(* IEC 61131-3 sources: SRCI/RobotLibrary/Library/POUs/AdvancedMove/MC_MoveCircularAbsolute, 1 file *)

(* ---- MC_MoveCircularAbsoluteFB.st ---- *)
/// Move the TCP to an absolute cartesian position (circular interpolation)
FUNCTION_BLOCK MC_MoveCircularAbsoluteFB EXTENDS RobotLibraryBaseExecuteFB
// -------------------------------------------------------------------------
//  SRCI Robot Library
// -------------------------------------------------------------------------
//
//  Object:      MoveCircularAbsoluteFB
//  Author:      Thorsten Brach
//  Date:        2024-06-01
//
//  Description:
//
//
//  Copyright:
//    (C) 2024 Thorsten Brach. All rights reserved
//             Licensed under the LGPL-3.0 license.
//
//  Disclaimer:
//    This project is provided without any guarantee and can be used for
//    private and commercial purposes. Any use is at the user’s
//    own risk and responsibility.
//
// -------------------------------------------------------------------------
VAR_INPUT
  /// Parameter which determines the behavior towards the previously sent and still active or buffered commands
  AbortingMode       : AbortingMode;
  /// Defines the target sequence in which the command will be executed
  SequenceFlag       : SequenceFlag;
  /// command results
  ParCmd             : MoveCircularAbsoluteParCmd;
END_VAR

VAR_OUTPUT
  /// Command is transferred and confirmed by the RC
  CommandBuffered    : BOOL;
  /// The command takes control of the motion of the according axis group
  Active             : BOOL;
  /// The command was aborted by another command.
  CommandAborted     : BOOL;
  /// TRUE, while command is interrupted during execution and can be continued
  CommandInterrupted : BOOL;
  /// command results
  OutCmd             : MoveCircularAbsoluteOutCmd;
END_VAR

VAR
  /// internal copy of command parameter
 _parCmd             : MoveCircularAbsoluteParCmd;
  /// command data to send
 _command            : MoveCircularAbsoluteSendData;
  /// response data received
 _response           : MoveCircularAbsoluteRecvData;
END_VAR

  SUPER^(AxesGroup := AxesGroup);

END_FUNCTION_BLOCK

METHOD INTERNAL CheckAddParameter : BOOL
VAR_INPUT
  /// Payload pointer
  PayloadPtr : UDINT;
END_VAR
VAR
  /// Payload as byte array
  Payload    : ARRAY [1..SIZEOF(_command)] OF BYTE;
  /// Null Byte array
  Null       : ARRAY [1..SIZEOF(_command)] OF BYTE;
  /// Data length to compare
  DataLen    : UDINT;
END_VAR

  // Payload pointer must be decreased by one byte, because ADR(Payload) is already one byte !
  PayloadPtr := LIMIT (0, PayloadPtr - 1, SIZEOF(Payload) -1);
  // Convert command struct to payload array
  SysDepMemCpy( pDest := ADR(Payload), pSrc := ADR(_command), DataLen := SIZEOF(_command));
  // Calculate the data length to compare - at least one byte must be compared !
  DataLen := LIMIT(1, SIZEOF(Payload) - PayloadPtr, SIZEOF(Payload));
  // Compare Payload-Array with Null-Byte-Array
  CheckAddParameter := SysDepMemCmp( pData1 := ADR(Payload) + PayloadPtr , pData2 := ADR(Null), DataLen := DataLen) <>  RobotLibraryConstants.OK ;

END_METHOD

METHOD PROTECTED CheckFunctionSupported : BOOL
VAR_IN_OUT
  /// Robot assignment of function
  AxesGroup : AxesGroup;
END_VAR

  CheckFunctionSupported := AxesGroup.State.RobotData.RCSupportedFunctions.MoveCircularAbsolute;

  IF ( NOT CheckFunctionSupported )
  THEN
    // call base implementation for set error and create log entry
    SUPER^.CheckFunctionSupported(AxesGroup := AxesGroup);
  END_IF

END_METHOD

METHOD PROTECTED CheckParameterChanged : BOOL
VAR_IN_OUT
  /// Robot assignment of function
  AxesGroup    : AxesGroup;
END_VAR

  // Check ParCmd Size is > 0, because MemCmp does not work correctly with size = 0
  IF (SIZEOF(ParCmd) = 0) OR (_stepCmd = 0)
  THEN
    RETURN;
  END_IF

  // compare memory
  _parameterChanged := ( SysDepMemCmp(pData1 := ADR(ParCmd), pData2 := ADR(_parCmd), DataLen := SIZEOF(ParCmd)) <> RobotLibraryConstants.OK );

  // check parameter valid ?
  _parameterValid   := CheckParameterValid( AxesGroup := AxesGroup );

  IF ((  _parameterChanged        )  AND
      (  _parameterValid          )) OR
      (  _parameterUpdateInternal )
  THEN
    // reset internal flag for send parameter update
   _parameterUpdateInternal := FALSE;
    // update internal copy of parameters
   _parCmd := ParCmd;
    // inc parameter sequence
   _command.ParSeq := _command.ParSeq + 1;
    // update command data
    CommandData := CreateCommandPayload(AxesGroup := AxesGroup); // ( Access via reference to rCommandFB in ACR )
    // notify active command register
    AxesGroup.Acyclic.ActiveCommandRegister.NotifyParameterChanged := _uniqueID;
  END_IF

END_METHOD

METHOD PROTECTED CheckParameterValid : BOOL
VAR_IN_OUT
  /// Robot assignment of function
  AxesGroup : AxesGroup;
END_VAR
VAR
  /// internal index for loops
 _idx : DINT;
END_VAR

  CheckParameterValid := TRUE;

  // Check AbortingMode valid ?
  IF (( AbortingMode <> AbortingModeEnum.BUFFER ) AND
      ( AbortingMode <> AbortingModeEnum.ABORT  ))
  THEN
    // Parameter not valid
    CheckParameterValid := FALSE;
    // Set error
    ErrorID := RobotLibraryErrorIdEnum.ERR_ABORTINGMODE_INVALID;
    // Create log entry
    CreateLogMessagePara1 ( Timestamp   := AxesGroup.State.SystemTime,
                            MessageType := MessageType.CMD,
                            Severity    := Severity.ERROR,
                            MessageCode := ErrorID,
                            MessageText := 'Invalid Parameter AbortingMode = {1}',
                            Para1       := ABORTING_MODE_TO_STRING(AbortingMode));
    RETURN;
  END_IF

  // Check SequenceFlag valid ?
  IF (( SequenceFlag <> SequenceFlagEnum.PRIMARY_SEQUENCE   ) AND
      ( SequenceFlag <> SequenceFlagEnum.SECONDARY_SEQUENCE ))
  THEN
    // Parameter not valid
    CheckParameterValid := FALSE;
    // Set error
    ErrorID := RobotLibraryErrorIdEnum.ERR_SEQFLAG_NOT_ALLOWED;
    // Create log entry
    CreateLogMessagePara1 ( Timestamp   := AxesGroup.State.SystemTime,
                            MessageType := MessageType.CMD,
                            Severity    := Severity.ERROR,
                            MessageCode := ErrorID,
                            MessageText := 'Invalid Parameter SequenceFlag = {1}',
                            Para1       := SEQUENCE_FLAG_TO_STRING(SequenceFlag));
    RETURN;
  END_IF

  // Check ParCmd.CircMode valid ?
  IF (( ParCmd.CircMode <> CircMode.BORDER            ) AND
      ( ParCmd.CircMode <> CircMode.CENTER            ) AND
      ( ParCmd.CircMode <> CircMode.CENTER_WITH_ANGLE ) AND
      ( ParCmd.CircMode <> CircMode.RADIUS            ))
  THEN
    // Parameter not valid
    CheckParameterValid := FALSE;
    // Set error
    ErrorID := RobotLibraryErrorIdEnum.ERR_INVALID_PAR_CMD;
    // Create log entry
    CreateLogMessagePara1 ( Timestamp   := AxesGroup.State.SystemTime,
                            MessageType := MessageType.CMD,
                            Severity    := Severity.ERROR,
                            MessageCode := ErrorID,
                            MessageText := 'Invalid Parameter ParCmd.CircMode = {1}',
                            Para1       :=  CIRC_MODE_TO_STRING(ParCmd.CircMode));
    RETURN;
  END_IF

  // Check ParCmd.AuxPoint.X valid ?
  IF ( SysDepIsValidReal(ParCmd.AuxPoint.X) = FALSE )
  THEN
    // Parameter not valid
    CheckParameterValid := FALSE;
    // Set error
    ErrorID := RobotLibraryErrorIdEnum.ERR_INVALID_PAR_CMD;

    // Create log entry
    CreateLogMessagePara1 ( Timestamp   := AxesGroup.State.SystemTime,
                            MessageType := MessageType.CMD,
                            Severity    := Severity.ERROR,
                            MessageCode := ErrorID,
                            MessageText := 'Invalid Parameter ParCmd.AuxPoint.X = {1}',
                            Para1       := VALID_REAL_TO_STRING(ParCmd.AuxPoint.X));
    RETURN;
  END_IF

  // Check ParCmd.AuxPoint.Y valid ?
  IF ( SysDepIsValidReal(ParCmd.AuxPoint.Y) = FALSE )
  THEN
    // Parameter not valid
    CheckParameterValid := FALSE;
    // Set error
    ErrorID := RobotLibraryErrorIdEnum.ERR_INVALID_PAR_CMD;

    // Create log entry
    CreateLogMessagePara1 ( Timestamp   := AxesGroup.State.SystemTime,
                            MessageType := MessageType.CMD,
                            Severity    := Severity.ERROR,
                            MessageCode := ErrorID,
                            MessageText := 'Invalid Parameter ParCmd.AuxPoint.Y = {1}',
                            Para1       := VALID_REAL_TO_STRING(ParCmd.AuxPoint.Y));
    RETURN;
  END_IF

  // Check ParCmd.AuxPoint.Z valid ?
  IF ( SysDepIsValidReal(ParCmd.AuxPoint.Z) = FALSE )
  THEN
    // Parameter not valid
    CheckParameterValid := FALSE;
    // Set error
    ErrorID := RobotLibraryErrorIdEnum.ERR_INVALID_PAR_CMD;

    // Create log entry
    CreateLogMessagePara1 ( Timestamp   := AxesGroup.State.SystemTime,
                            MessageType := MessageType.CMD,
                            Severity    := Severity.ERROR,
                            MessageCode := ErrorID,
                            MessageText := 'Invalid Parameter ParCmd.AuxPoint.Z = {1}',
                            Para1       := VALID_REAL_TO_STRING(ParCmd.AuxPoint.Z));
    RETURN;
  END_IF

  // Check ParCmd.AuxPoint.Rx valid ?
  IF ( SysDepIsValidReal(ParCmd.AuxPoint.Rx) = FALSE )
  THEN
    // Parameter not valid
    CheckParameterValid := FALSE;
    // Set error
    ErrorID := RobotLibraryErrorIdEnum.ERR_INVALID_PAR_CMD;

    // Create log entry
    CreateLogMessagePara1 ( Timestamp   := AxesGroup.State.SystemTime,
                            MessageType := MessageType.CMD,
                            Severity    := Severity.ERROR,
                            MessageCode := ErrorID,
                            MessageText := 'Invalid Parameter ParCmd.AuxPoint.Rx = {1}',
                            Para1       := VALID_REAL_TO_STRING(ParCmd.AuxPoint.Rx));
    RETURN;
  END_IF

  // Check ParCmd.AuxPoint.Ry valid ?
  IF ( SysDepIsValidReal(ParCmd.AuxPoint.Ry) = FALSE )
  THEN
    // Parameter not valid
    CheckParameterValid := FALSE;
    // Set error
    ErrorID := RobotLibraryErrorIdEnum.ERR_INVALID_PAR_CMD;

    // Create log entry
    CreateLogMessagePara1 ( Timestamp   := AxesGroup.State.SystemTime,
                            MessageType := MessageType.CMD,
                            Severity    := Severity.ERROR,
                            MessageCode := ErrorID,
                            MessageText := 'Invalid Parameter ParCmd.AuxPoint.Ry = {1}',
                            Para1       := VALID_REAL_TO_STRING(ParCmd.AuxPoint.Ry));
    RETURN;
  END_IF

  // Check ParCmd.AuxPoint.Rz valid ?
  IF ( SysDepIsValidReal(ParCmd.AuxPoint.Rz) = FALSE )
  THEN
    // Parameter not valid
    CheckParameterValid := FALSE;
    // Set error
    ErrorID := RobotLibraryErrorIdEnum.ERR_INVALID_PAR_CMD;

    // Create log entry
    CreateLogMessagePara1 ( Timestamp   := AxesGroup.State.SystemTime,
                            MessageType := MessageType.CMD,
                            Severity    := Severity.ERROR,
                            MessageCode := ErrorID,
                            MessageText := 'Invalid Parameter ParCmd.AuxPoint.Rz = {1}',
                            Para1       := VALID_REAL_TO_STRING(ParCmd.AuxPoint.Rz));
    RETURN;
  END_IF

  // Check ParCmd.AuxPoint.E1 valid ?
  IF ( SysDepIsValidReal(ParCmd.AuxPoint.E1) = FALSE )
  THEN
    // Parameter not valid
    CheckParameterValid := FALSE;
    // Set error
    ErrorID := RobotLibraryErrorIdEnum.ERR_INVALID_PAR_CMD;

    // Create log entry
    CreateLogMessagePara1 ( Timestamp   := AxesGroup.State.SystemTime,
                            MessageType := MessageType.CMD,
                            Severity    := Severity.ERROR,
                            MessageCode := ErrorID,
                            MessageText := 'Invalid Parameter ParCmd.AuxPoint.E1 = {1}',
                            Para1       := VALID_REAL_TO_STRING(ParCmd.AuxPoint.E1));
    RETURN;
  END_IF

  // Check ParCmd.AuxPoint.E2 valid ?
  IF ( SysDepIsValidReal(ParCmd.AuxPoint.E2) = FALSE )
  THEN
    // Parameter not valid
    CheckParameterValid := FALSE;
    // Set error
    ErrorID := RobotLibraryErrorIdEnum.ERR_INVALID_PAR_CMD;

    // Create log entry
    CreateLogMessagePara1 ( Timestamp   := AxesGroup.State.SystemTime,
                            MessageType := MessageType.CMD,
                            Severity    := Severity.ERROR,
                            MessageCode := ErrorID,
                            MessageText := 'Invalid Parameter ParCmd.AuxPoint.E2 = {1}',
                            Para1       := VALID_REAL_TO_STRING(ParCmd.AuxPoint.E2));
    RETURN;
  END_IF

  // Check ParCmd.AuxPoint.E3 valid ?
  IF ( SysDepIsValidReal(ParCmd.AuxPoint.E3) = FALSE )
  THEN
    // Parameter not valid
    CheckParameterValid := FALSE;
    // Set error
    ErrorID := RobotLibraryErrorIdEnum.ERR_INVALID_PAR_CMD;

    // Create log entry
    CreateLogMessagePara1 ( Timestamp   := AxesGroup.State.SystemTime,
                            MessageType := MessageType.CMD,
                            Severity    := Severity.ERROR,
                            MessageCode := ErrorID,
                            MessageText := 'Invalid Parameter ParCmd.AuxPoint.E3 = {1}',
                            Para1       := VALID_REAL_TO_STRING(ParCmd.AuxPoint.E3));
    RETURN;
  END_IF

  // Check ParCmd.AuxPoint.E4 valid ?
  IF ( SysDepIsValidReal(ParCmd.AuxPoint.E4) = FALSE )
  THEN
    // Parameter not valid
    CheckParameterValid := FALSE;
    // Set error
    ErrorID := RobotLibraryErrorIdEnum.ERR_INVALID_PAR_CMD;

    // Create log entry
    CreateLogMessagePara1 ( Timestamp   := AxesGroup.State.SystemTime,
                            MessageType := MessageType.CMD,
                            Severity    := Severity.ERROR,
                            MessageCode := ErrorID,
                            MessageText := 'Invalid Parameter ParCmd.AuxPoint.E4 = {1}',
                            Para1       := VALID_REAL_TO_STRING(ParCmd.AuxPoint.E4));
    RETURN;
  END_IF

  // Check ParCmd.AuxPoint.E5 valid ?
  IF ( SysDepIsValidReal(ParCmd.AuxPoint.E5) = FALSE )
  THEN
    // Parameter not valid
    CheckParameterValid := FALSE;
    // Set error
    ErrorID := RobotLibraryErrorIdEnum.ERR_INVALID_PAR_CMD;

    // Create log entry
    CreateLogMessagePara1 ( Timestamp   := AxesGroup.State.SystemTime,
                            MessageType := MessageType.CMD,
                            Severity    := Severity.ERROR,
                            MessageCode := ErrorID,
                            MessageText := 'Invalid Parameter ParCmd.AuxPoint.E5 = {1}',
                            Para1       := VALID_REAL_TO_STRING(ParCmd.AuxPoint.E5));
    RETURN;
  END_IF

  // Check ParCmd.AuxPoint.E6 valid ?
  IF ( SysDepIsValidReal(ParCmd.AuxPoint.E6) = FALSE )
  THEN
    // Parameter not valid
    CheckParameterValid := FALSE;
    // Set error
    ErrorID := RobotLibraryErrorIdEnum.ERR_INVALID_PAR_CMD;

    // Create log entry
    CreateLogMessagePara1 ( Timestamp   := AxesGroup.State.SystemTime,
                            MessageType := MessageType.CMD,
                            Severity    := Severity.ERROR,
                            MessageCode := ErrorID,
                            MessageText := 'Invalid Parameter ParCmd.AuxPoint.E6 = {1}',
                            Para1       := VALID_REAL_TO_STRING(ParCmd.AuxPoint.E6));
    RETURN;
  END_IF

  // Check ParCmd.AuxPoint.Config.Shoulder valid ?
  IF (( ParCmd.AuxPoint.Config.Shoulder <> ArmConfigShoulder.USE_CONFIG ) AND
      ( ParCmd.AuxPoint.Config.Shoulder <> ArmConfigShoulder.SAME       ) AND
      ( ParCmd.AuxPoint.Config.Shoulder <> ArmConfigShoulder.FREE       ) AND
      ( ParCmd.AuxPoint.Config.Shoulder <> ArmConfigShoulder.BACK       ) AND
      ( ParCmd.AuxPoint.Config.Shoulder <> ArmConfigShoulder.FRONT      ))
  THEN
    // Parameter not valid
    CheckParameterValid := FALSE;
    // Set error
    ErrorID := RobotLibraryErrorIdEnum.ERR_CONFIGMODE_SHOULDER_INVALID;
    // Create log entry
    CreateLogMessagePara1 ( Timestamp   := AxesGroup.State.SystemTime,
                            MessageType := MessageType.CMD,
                            Severity    := Severity.ERROR,
                            MessageCode := ErrorID,
                            MessageText := 'Invalid Parameter ParCmd.AuxPoint.Config.Shoulder = {1}',
                            Para1       :=  ARM_CONFIG_SHOULDER_TO_STRING(ParCmd.AuxPoint.Config.Shoulder));
    RETURN;
  END_IF

  // Check ParCmd.AuxPoint.Config.Elbow valid ?
  IF (( ParCmd.AuxPoint.Config.Elbow <> ArmConfigElbow.USE_CONFIG ) AND
      ( ParCmd.AuxPoint.Config.Elbow <> ArmConfigElbow.SAME       ) AND
      ( ParCmd.AuxPoint.Config.Elbow <> ArmConfigElbow.FREE       ) AND
      ( ParCmd.AuxPoint.Config.Elbow <> ArmConfigElbow.DOWN       ) AND
      ( ParCmd.AuxPoint.Config.Elbow <> ArmConfigElbow.UP         ))
  THEN
    // Parameter not valid
    CheckParameterValid := FALSE;
    // Set error
    ErrorID := RobotLibraryErrorIdEnum.ERR_CONFIGMODE_ELBOW_INVALID;
    // Create log entry
    CreateLogMessagePara1 ( Timestamp   := AxesGroup.State.SystemTime,
                            MessageType := MessageType.CMD,
                            Severity    := Severity.ERROR,
                            MessageCode := ErrorID,
                            MessageText := 'Invalid Parameter ParCmd.AuxPoint.Config.Elbow = {1}',
                            Para1       :=  ARM_CONFIG_ELBOW_TO_STRING(ParCmd.AuxPoint.Config.Elbow));
    RETURN;
  END_IF

  // Check ParCmd.AuxPoint.Config.Wrist valid ?
  IF (( ParCmd.AuxPoint.Config.Wrist <> ArmConfigWrist.USE_CONFIG ) AND
      ( ParCmd.AuxPoint.Config.Wrist <> ArmConfigWrist.SAME       ) AND
      ( ParCmd.AuxPoint.Config.Wrist <> ArmConfigWrist.FREE       ) AND
      ( ParCmd.AuxPoint.Config.Wrist <> ArmConfigWrist.FLIP       ) AND
      ( ParCmd.AuxPoint.Config.Wrist <> ArmConfigWrist.NON_FLIP   ))
  THEN
    // Parameter not valid
    CheckParameterValid := FALSE;
    // Set error
    ErrorID := RobotLibraryErrorIdEnum.ERR_CONFIGMODE_WRIST_INVALID;
    // Create log entry
    CreateLogMessagePara1 ( Timestamp   := AxesGroup.State.SystemTime,
                            MessageType := MessageType.CMD,
                            Severity    := Severity.ERROR,
                            MessageCode := ErrorID,
                            MessageText := 'Invalid Parameter ParCmd.AuxPoint.Config.Wrist = {1}',
                            Para1       :=  ARM_CONFIG_WRIST_TO_STRING(ParCmd.AuxPoint.Config.Wrist));
    RETURN;
  END_IF

  // Check ParCmd.CircPlane valid ?
  IF (( ParCmd.CircPlane <> CircPlane.XZ_PLANE ) AND
      ( ParCmd.CircPlane <> CircPlane.YZ_PLANE ) AND
      ( ParCmd.CircPlane <> CircPlane.XY_PLANE ))
  THEN
    // Parameter not valid
    CheckParameterValid := FALSE;
    // Set error
    ErrorID := RobotLibraryErrorIdEnum.ERR_INVALID_PAR_CMD;
    // Create log entry
    CreateLogMessagePara1 ( Timestamp   := AxesGroup.State.SystemTime,
                            MessageType := MessageType.CMD,
                            Severity    := Severity.ERROR,
                            MessageCode := ErrorID,
                            MessageText := 'Invalid Parameter ParCmd.CircPlane = {1}',
                            Para1       :=  CIRC_PLANE_TO_STRING(ParCmd.CircPlane));
    RETURN;
  END_IF

  // Check ParCmd.Tolerance valid ?
  IF ( SysDepIsValidReal(ParCmd.Tolerance) = FALSE )
  THEN
    // Parameter not valid
    CheckParameterValid := FALSE;
    // Set error
    ErrorID := RobotLibraryErrorIdEnum.ERR_INVALID_PAR_CMD;

    // Create log entry
    CreateLogMessagePara1 ( Timestamp   := AxesGroup.State.SystemTime,
                            MessageType := MessageType.CMD,
                            Severity    := Severity.ERROR,
                            MessageCode := ErrorID,
                            MessageText := 'Invalid Parameter ParCmd.Tolerance = {1}',
                            Para1       := VALID_REAL_TO_STRING(ParCmd.Tolerance));
    RETURN;
  END_IF

  // Check ParCmd.EndPoint.X valid ?
  IF ( SysDepIsValidReal(ParCmd.EndPoint.X) = FALSE )
  THEN
    // Parameter not valid
    CheckParameterValid := FALSE;
    // Set error
    ErrorID := RobotLibraryErrorIdEnum.ERR_INVALID_PAR_CMD;

    // Create log entry
    CreateLogMessagePara1 ( Timestamp   := AxesGroup.State.SystemTime,
                            MessageType := MessageType.CMD,
                            Severity    := Severity.ERROR,
                            MessageCode := ErrorID,
                            MessageText := 'Invalid Parameter ParCmd.EndPoint.X = {1}',
                            Para1       := VALID_REAL_TO_STRING(ParCmd.EndPoint.X));
    RETURN;
  END_IF

  // Check ParCmd.EndPoint.Y valid ?
  IF ( SysDepIsValidReal(ParCmd.EndPoint.Y) = FALSE )
  THEN
    // Parameter not valid
    CheckParameterValid := FALSE;
    // Set error
    ErrorID := RobotLibraryErrorIdEnum.ERR_INVALID_PAR_CMD;

    // Create log entry
    CreateLogMessagePara1 ( Timestamp   := AxesGroup.State.SystemTime,
                            MessageType := MessageType.CMD,
                            Severity    := Severity.ERROR,
                            MessageCode := ErrorID,
                            MessageText := 'Invalid Parameter ParCmd.EndPoint.Y = {1}',
                            Para1       := VALID_REAL_TO_STRING(ParCmd.EndPoint.Y));
    RETURN;
  END_IF

  // Check ParCmd.EndPoint.Z valid ?
  IF ( SysDepIsValidReal(ParCmd.EndPoint.Z) = FALSE )
  THEN
    // Parameter not valid
    CheckParameterValid := FALSE;
    // Set error
    ErrorID := RobotLibraryErrorIdEnum.ERR_INVALID_PAR_CMD;

    // Create log entry
    CreateLogMessagePara1 ( Timestamp   := AxesGroup.State.SystemTime,
                            MessageType := MessageType.CMD,
                            Severity    := Severity.ERROR,
                            MessageCode := ErrorID,
                            MessageText := 'Invalid Parameter ParCmd.EndPoint.Z = {1}',
                            Para1       := VALID_REAL_TO_STRING(ParCmd.EndPoint.Z));
    RETURN;
  END_IF

  // Check ParCmd.EndPoint.Rx valid ?
  IF ( SysDepIsValidReal(ParCmd.EndPoint.Rx) = FALSE )
  THEN
    // Parameter not valid
    CheckParameterValid := FALSE;
    // Set error
    ErrorID := RobotLibraryErrorIdEnum.ERR_INVALID_PAR_CMD;

    // Create log entry
    CreateLogMessagePara1 ( Timestamp   := AxesGroup.State.SystemTime,
                            MessageType := MessageType.CMD,
                            Severity    := Severity.ERROR,
                            MessageCode := ErrorID,
                            MessageText := 'Invalid Parameter ParCmd.EndPoint.Rx = {1}',
                            Para1       := VALID_REAL_TO_STRING(ParCmd.EndPoint.Rx));
    RETURN;
  END_IF

  // Check ParCmd.EndPoint.Ry valid ?
  IF ( SysDepIsValidReal(ParCmd.EndPoint.Ry) = FALSE )
  THEN
    // Parameter not valid
    CheckParameterValid := FALSE;
    // Set error
    ErrorID := RobotLibraryErrorIdEnum.ERR_INVALID_PAR_CMD;

    // Create log entry
    CreateLogMessagePara1 ( Timestamp   := AxesGroup.State.SystemTime,
                            MessageType := MessageType.CMD,
                            Severity    := Severity.ERROR,
                            MessageCode := ErrorID,
                            MessageText := 'Invalid Parameter ParCmd.EndPoint.Ry = {1}',
                            Para1       := VALID_REAL_TO_STRING(ParCmd.EndPoint.Ry));
    RETURN;
  END_IF

  // Check ParCmd.EndPoint.Rz valid ?
  IF ( SysDepIsValidReal(ParCmd.EndPoint.Rz) = FALSE )
  THEN
    // Parameter not valid
    CheckParameterValid := FALSE;
    // Set error
    ErrorID := RobotLibraryErrorIdEnum.ERR_INVALID_PAR_CMD;

    // Create log entry
    CreateLogMessagePara1 ( Timestamp   := AxesGroup.State.SystemTime,
                            MessageType := MessageType.CMD,
                            Severity    := Severity.ERROR,
                            MessageCode := ErrorID,
                            MessageText := 'Invalid Parameter ParCmd.EndPoint.Rz = {1}',
                            Para1       := VALID_REAL_TO_STRING(ParCmd.EndPoint.Rz));
    RETURN;
  END_IF

  // Check ParCmd.EndPoint.E1 valid ?
  IF ( SysDepIsValidReal(ParCmd.EndPoint.E1) = FALSE )
  THEN
    // Parameter not valid
    CheckParameterValid := FALSE;
    // Set error
    ErrorID := RobotLibraryErrorIdEnum.ERR_INVALID_PAR_CMD;

    // Create log entry
    CreateLogMessagePara1 ( Timestamp   := AxesGroup.State.SystemTime,
                            MessageType := MessageType.CMD,
                            Severity    := Severity.ERROR,
                            MessageCode := ErrorID,
                            MessageText := 'Invalid Parameter ParCmd.EndPoint.E1 = {1}',
                            Para1       := VALID_REAL_TO_STRING(ParCmd.EndPoint.E1));
    RETURN;
  END_IF

  // Check ParCmd.EndPoint.E2 valid ?
  IF ( SysDepIsValidReal(ParCmd.EndPoint.E2) = FALSE )
  THEN
    // Parameter not valid
    CheckParameterValid := FALSE;
    // Set error
    ErrorID := RobotLibraryErrorIdEnum.ERR_INVALID_PAR_CMD;

    // Create log entry
    CreateLogMessagePara1 ( Timestamp   := AxesGroup.State.SystemTime,
                            MessageType := MessageType.CMD,
                            Severity    := Severity.ERROR,
                            MessageCode := ErrorID,
                            MessageText := 'Invalid Parameter ParCmd.EndPoint.E2 = {1}',
                            Para1       := VALID_REAL_TO_STRING(ParCmd.EndPoint.E2));
    RETURN;
  END_IF

  // Check ParCmd.EndPoint.E3 valid ?
  IF ( SysDepIsValidReal(ParCmd.EndPoint.E3) = FALSE )
  THEN
    // Parameter not valid
    CheckParameterValid := FALSE;
    // Set error
    ErrorID := RobotLibraryErrorIdEnum.ERR_INVALID_PAR_CMD;

    // Create log entry
    CreateLogMessagePara1 ( Timestamp   := AxesGroup.State.SystemTime,
                            MessageType := MessageType.CMD,
                            Severity    := Severity.ERROR,
                            MessageCode := ErrorID,
                            MessageText := 'Invalid Parameter ParCmd.EndPoint.E3 = {1}',
                            Para1       := VALID_REAL_TO_STRING(ParCmd.EndPoint.E3));
    RETURN;
  END_IF

  // Check ParCmd.EndPoint.E4 valid ?
  IF ( SysDepIsValidReal(ParCmd.EndPoint.E4) = FALSE )
  THEN
    // Parameter not valid
    CheckParameterValid := FALSE;
    // Set error
    ErrorID := RobotLibraryErrorIdEnum.ERR_INVALID_PAR_CMD;

    // Create log entry
    CreateLogMessagePara1 ( Timestamp   := AxesGroup.State.SystemTime,
                            MessageType := MessageType.CMD,
                            Severity    := Severity.ERROR,
                            MessageCode := ErrorID,
                            MessageText := 'Invalid Parameter ParCmd.EndPoint.E4 = {1}',
                            Para1       := VALID_REAL_TO_STRING(ParCmd.EndPoint.E4));
    RETURN;
  END_IF

  // Check ParCmd.EndPoint.E5 valid ?
  IF ( SysDepIsValidReal(ParCmd.EndPoint.E5) = FALSE )
  THEN
    // Parameter not valid
    CheckParameterValid := FALSE;
    // Set error
    ErrorID := RobotLibraryErrorIdEnum.ERR_INVALID_PAR_CMD;

    // Create log entry
    CreateLogMessagePara1 ( Timestamp   := AxesGroup.State.SystemTime,
                            MessageType := MessageType.CMD,
                            Severity    := Severity.ERROR,
                            MessageCode := ErrorID,
                            MessageText := 'Invalid Parameter ParCmd.EndPoint.E5 = {1}',
                            Para1       := VALID_REAL_TO_STRING(ParCmd.EndPoint.E5));
    RETURN;
  END_IF

  // Check ParCmd.EndPoint.E6 valid ?
  IF ( SysDepIsValidReal(ParCmd.EndPoint.E6) = FALSE )
  THEN
    // Parameter not valid
    CheckParameterValid := FALSE;
    // Set error
    ErrorID := RobotLibraryErrorIdEnum.ERR_INVALID_PAR_CMD;

    // Create log entry
    CreateLogMessagePara1 ( Timestamp   := AxesGroup.State.SystemTime,
                            MessageType := MessageType.CMD,
                            Severity    := Severity.ERROR,
                            MessageCode := ErrorID,
                            MessageText := 'Invalid Parameter ParCmd.EndPoint.E6 = {1}',
                            Para1       := VALID_REAL_TO_STRING(ParCmd.EndPoint.E6));
    RETURN;
  END_IF

  // Check ParCmd.EndPoint.Config.Shoulder valid ?
  IF (( ParCmd.EndPoint.Config.Shoulder <> ArmConfigShoulder.USE_CONFIG ) AND
      ( ParCmd.EndPoint.Config.Shoulder <> ArmConfigShoulder.SAME       ) AND
      ( ParCmd.EndPoint.Config.Shoulder <> ArmConfigShoulder.FREE       ) AND
      ( ParCmd.EndPoint.Config.Shoulder <> ArmConfigShoulder.BACK       ) AND
      ( ParCmd.EndPoint.Config.Shoulder <> ArmConfigShoulder.FRONT      ))
  THEN
    // Parameter not valid
    CheckParameterValid := FALSE;
    // Set error
    ErrorID := RobotLibraryErrorIdEnum.ERR_CONFIGMODE_SHOULDER_INVALID;
    // Create log entry
    CreateLogMessagePara1 ( Timestamp   := AxesGroup.State.SystemTime,
                            MessageType := MessageType.CMD,
                            Severity    := Severity.ERROR,
                            MessageCode := ErrorID,
                            MessageText := 'Invalid Parameter ParCmd.EndPoint.Config.Shoulder = {1}',
                            Para1       :=  ARM_CONFIG_SHOULDER_TO_STRING(ParCmd.EndPoint.Config.Shoulder));
    RETURN;
  END_IF

  // Check ParCmd.EndPoint.Config.Elbow valid ?
  IF (( ParCmd.EndPoint.Config.Elbow <> ArmConfigElbow.USE_CONFIG ) AND
      ( ParCmd.EndPoint.Config.Elbow <> ArmConfigElbow.SAME       ) AND
      ( ParCmd.EndPoint.Config.Elbow <> ArmConfigElbow.FREE       ) AND
      ( ParCmd.EndPoint.Config.Elbow <> ArmConfigElbow.DOWN       ) AND
      ( ParCmd.EndPoint.Config.Elbow <> ArmConfigElbow.UP         ))
  THEN
    // Parameter not valid
    CheckParameterValid := FALSE;
    // Set error
    ErrorID := RobotLibraryErrorIdEnum.ERR_CONFIGMODE_ELBOW_INVALID;
    // Create log entry
    CreateLogMessagePara1 ( Timestamp   := AxesGroup.State.SystemTime,
                            MessageType := MessageType.CMD,
                            Severity    := Severity.ERROR,
                            MessageCode := ErrorID,
                            MessageText := 'Invalid Parameter ParCmd.EndPoint.Config.Elbow = {1}',
                            Para1       :=  ARM_CONFIG_ELBOW_TO_STRING(ParCmd.EndPoint.Config.Elbow));
    RETURN;
  END_IF

  // Check ParCmd.EndPoint.Config.Wrist valid ?
  IF (( ParCmd.EndPoint.Config.Wrist <> ArmConfigWrist.USE_CONFIG ) AND
      ( ParCmd.EndPoint.Config.Wrist <> ArmConfigWrist.SAME       ) AND
      ( ParCmd.EndPoint.Config.Wrist <> ArmConfigWrist.FREE       ) AND
      ( ParCmd.EndPoint.Config.Wrist <> ArmConfigWrist.FLIP       ) AND
      ( ParCmd.EndPoint.Config.Wrist <> ArmConfigWrist.NON_FLIP   ))
  THEN
    // Parameter not valid
    CheckParameterValid := FALSE;
    // Set error
    ErrorID := RobotLibraryErrorIdEnum.ERR_CONFIGMODE_WRIST_INVALID;
    // Create log entry
    CreateLogMessagePara1 ( Timestamp   := AxesGroup.State.SystemTime,
                            MessageType := MessageType.CMD,
                            Severity    := Severity.ERROR,
                            MessageCode := ErrorID,
                            MessageText := 'Invalid Parameter ParCmd.EndPoint.Config.Wrist = {1}',
                            Para1       :=  ARM_CONFIG_WRIST_TO_STRING(ParCmd.EndPoint.Config.Wrist));
    RETURN;
  END_IF

  // Check ParCmd.Angle valid ?
  IF ( SysDepIsValidReal(ParCmd.Angle) = FALSE )
  THEN
    // Parameter not valid
    CheckParameterValid := FALSE;
    // Set error
    ErrorID := RobotLibraryErrorIdEnum.ERR_INVALID_PAR_CMD;

    // Create log entry
    CreateLogMessagePara1 ( Timestamp   := AxesGroup.State.SystemTime,
                            MessageType := MessageType.CMD,
                            Severity    := Severity.ERROR,
                            MessageCode := ErrorID,
                            MessageText := 'Invalid Parameter ParCmd.Angle = {1}',
                            Para1       := VALID_REAL_TO_STRING(ParCmd.Angle));
    RETURN;
  END_IF

  // Check ParCmd.PathChoice valid ?
  IF (( ParCmd.PathChoice <> PathChoice.CLOCKWISE  ) AND
      ( ParCmd.PathChoice <> PathChoice.COUNTERCLOCKWISE ))
  THEN
    // Parameter not valid
    CheckParameterValid := FALSE;
    // Set error
    ErrorID := RobotLibraryErrorIdEnum.ERR_INVALID_PAR_CMD;
    // Create log entry
    CreateLogMessagePara1 ( Timestamp   := AxesGroup.State.SystemTime,
                            MessageType := MessageType.CMD,
                            Severity    := Severity.ERROR,
                            MessageCode := ErrorID,
                            MessageText := 'Invalid Parameter ParCmd.PathChoice = {1}',
                            Para1       := PATH_CHOICE_TO_STRING(ParCmd.PathChoice));
    RETURN;
  END_IF

  // Check ParCmd.VelocityRate valid ?
  IF  (( SysDepIsValidReal(ParCmd.VelocityRate) = FALSE )  OR
      ((                   ParCmd.VelocityRate  <     0 )  AND
       (                   ParCmd.VelocityRate <>    -1 )) OR
       (                   ParCmd.VelocityRate  >   100 ))
  THEN
    // Parameter not valid
    CheckParameterValid := FALSE;
    // Set error
    ErrorID := RobotLibraryErrorIdEnum.ERR_VELOCITY_INVALID;
    // Create log entry
    CreateLogMessagePara1 ( Timestamp   := AxesGroup.State.SystemTime,
                            MessageType := MessageType.CMD,
                            Severity    := Severity.ERROR,
                            MessageCode := ErrorID,
                            MessageText := 'Invalid Parameter ParCmd.VelocityRate = {1}',
                            Para1       := VALID_REAL_TO_STRING(ParCmd.VelocityRate));
    RETURN;
  END_IF

  // Check ParCmd.AccelerationRate valid ?
  IF  (( SysDepIsValidReal(ParCmd.AccelerationRate) = FALSE )  OR
      ((                   ParCmd.AccelerationRate  <     0 )  AND
       (                   ParCmd.AccelerationRate <>    -1 )) OR
       (                   ParCmd.AccelerationRate  >   100 ))
  THEN
    // Parameter not valid
    CheckParameterValid := FALSE;
    // Set error
    ErrorID := RobotLibraryErrorIdEnum.ERR_ACCELERATION_INVALID;
    // Create log entry
    CreateLogMessagePara1 ( Timestamp   := AxesGroup.State.SystemTime,
                            MessageType := MessageType.CMD,
                            Severity    := Severity.ERROR,
                            MessageCode := ErrorID,
                            MessageText := 'Invalid Parameter ParCmd.AccelerationRate = {1}',
                            Para1       := VALID_REAL_TO_STRING(ParCmd.AccelerationRate));
    RETURN;
  END_IF

  // Check ParCmd.DecelerationRate valid ?
  IF  (( SysDepIsValidReal(ParCmd.DecelerationRate) = FALSE )  OR
      ((                   ParCmd.DecelerationRate  <     0 )  AND
       (                   ParCmd.DecelerationRate <>    -1 )) OR
       (                   ParCmd.DecelerationRate  >   100 ))
  THEN
    // Parameter not valid
    CheckParameterValid := FALSE;
    // Set error
    ErrorID := RobotLibraryErrorIdEnum.ERR_DECELERATION_INVALID;
    // Create log entry
    CreateLogMessagePara1 ( Timestamp   := AxesGroup.State.SystemTime,
                            MessageType := MessageType.CMD,
                            Severity    := Severity.ERROR,
                            MessageCode := ErrorID,
                            MessageText := 'Invalid Parameter ParCmd.DecelerationRate = {1}',
                            Para1       := VALID_REAL_TO_STRING(ParCmd.DecelerationRate));
    RETURN;
  END_IF

  // Check ParCmd.JerkRate valid ?
  IF  (( SysDepIsValidReal(ParCmd.JerkRate) = FALSE )  OR
      ((                   ParCmd.JerkRate  <     0 )  AND
       (                   ParCmd.JerkRate <>    -1 )) OR
       (                   ParCmd.JerkRate  >   100 ))
  THEN
    // Parameter not valid
    CheckParameterValid := FALSE;
    // Set error
    ErrorID := RobotLibraryErrorIdEnum.ERR_JERK_INVALID;
    // Create log entry
    CreateLogMessagePara1 ( Timestamp   := AxesGroup.State.SystemTime,
                            MessageType := MessageType.CMD,
                            Severity    := Severity.ERROR,
                            MessageCode := ErrorID,
                            MessageText := 'Invalid Parameter ParCmd.JerkRate = {1}',
                            Para1       := VALID_REAL_TO_STRING(ParCmd.JerkRate));
    RETURN;
  END_IF

  // Check ParCmd.ToolNo valid ?
  IF (( ParCmd.ToolNo <   0                                                ) OR
      ( ParCmd.ToolNo > 254                                                ) OR
      ( ParCmd.ToolNo > AxesGroup.State.ConfigurationData.HighestToolIndex ) OR
      ( ParCmd.ToolNo > RobotLibraryParameter.TOOL_MAX -1                  ))
  THEN
    // Parameter not valid
    CheckParameterValid := FALSE;

    // Check ToolNo available on RC ?
    IF ( ParCmd.ToolNo > AxesGroup.State.ConfigurationData.HighestToolIndex )
    THEN
      ErrorID := RobotLibraryErrorIdEnum.ERR_TOOLNO_UNAVAILABLE;
    ELSE
      ErrorID := RobotLibraryErrorIdEnum.ERR_TOOLNO_RANGE;
  	END_IF

    // Create log entry
    CreateLogMessagePara1 ( Timestamp   := AxesGroup.State.SystemTime,
                            MessageType := MessageType.CMD,
                            Severity    := Severity.ERROR,
                            MessageCode := ErrorID,
                            MessageText := 'Invalid Parameter ParCmd.ToolNo = {1}',
                            Para1       := USINT_TO_STRING(ParCmd.ToolNo));
    RETURN;
  END_IF

  // Check ParCmd.FrameNo valid ?
  IF (( ParCmd.FrameNo <   0                                                 ) OR
      ( ParCmd.FrameNo > 254                                                 ) OR
      ( ParCmd.FrameNo > AxesGroup.State.ConfigurationData.HighestFrameIndex ) OR
      ( ParCmd.FrameNo > RobotLibraryParameter.FRAME_MAX -1                  ))
  THEN
    // Parameter not valid
    CheckParameterValid := FALSE;

    // Check FrameNo available on RC ?
    IF ( ParCmd.FrameNo > AxesGroup.State.ConfigurationData.HighestFrameIndex )
    THEN
      ErrorID := RobotLibraryErrorIdEnum.ERR_FRAMENO_UNAVAILABLE;
    ELSE
      ErrorID := RobotLibraryErrorIdEnum.ERR_FRAMENO_RANGE;
  	END_IF

    // Create log entry
    CreateLogMessagePara1 ( Timestamp   := AxesGroup.State.SystemTime,
                            MessageType := MessageType.CMD,
                            Severity    := Severity.ERROR,
                            MessageCode := ErrorID,
                            MessageText := 'Invalid Parameter ParCmd.FrameNo = {1}',
                            Para1       := USINT_TO_STRING(ParCmd.FrameNo));
    RETURN;
  END_IF

  // Check ParCmd.BlendingMode valid ?
  IF (( ParCmd.BlendingMode <> BlendingMode.EXACT_STOP           ) AND
      ( ParCmd.BlendingMode <> BlendingMode.DEFINED_VELOCITY     ) AND
      ( ParCmd.BlendingMode <> BlendingMode.CORNER_DISTANCE      ) AND
      ( ParCmd.BlendingMode <> BlendingMode.MAX_CORNER_DEVIATION ) AND
      ( ParCmd.BlendingMode <> BlendingMode.CORNER_DISTANCE_2R   ) AND
      ( ParCmd.BlendingMode <> BlendingMode.RAMP_OVERLAP         ) AND
      ( ParCmd.BlendingMode <> BlendingMode.CORNER_DISTANCE_1R   ))
  THEN
    // Parameter not valid
    CheckParameterValid := FALSE;
    // Set error
    ErrorID := RobotLibraryErrorIdEnum.ERR_INVALID_PAR_CMD;
    // Create log entry
    CreateLogMessagePara1 ( Timestamp   := AxesGroup.State.SystemTime,
                            MessageType := MessageType.CMD,
                            Severity    := Severity.ERROR,
                            MessageCode := ErrorID,
                            MessageText := 'Invalid Parameter ParCmd.BlendingMode = {1}',
                            Para1       := BLENDING_MODE_TO_STRING(ParCmd.BlendingMode));
    RETURN;
  END_IF

  FOR _idx := 0 TO 1
  DO
    // Check ParCmd.BlendingParameter valid ?
    IF  ( SysDepIsValidReal(ParCmd.BlendingParameter[_idx]) = FALSE )
    THEN
      // Parameter not valid
      CheckParameterValid := FALSE;
      // Set error
      ErrorID := RobotLibraryErrorIdEnum.ERR_JERK_INVALID;
      // Create log entry
      CreateLogMessagePara2 ( Timestamp   := AxesGroup.State.SystemTime,
                              MessageType := MessageType.CMD,
                              Severity    := Severity.ERROR,
                              MessageCode := ErrorID,
                              MessageText := 'Invalid Parameter ParCmd.BlendingParameter[{2}] = {1}',
                              Para1       := VALID_REAL_TO_STRING(ParCmd.JerkRate),
                              Para2       := DINT_TO_STRING(_idx));
      EXIT;
      RETURN;
    END_IF
  END_FOR

  // Check ParCmd.MoveTime valid ?
  IF  ( ParCmd.MoveTime < T#0S )
  THEN
    // Parameter not valid
    CheckParameterValid := FALSE;
    // Set error
    ErrorID := RobotLibraryErrorIdEnum.ERR_INVALID_PAR_CMD;
    // Create log entry
    CreateLogMessagePara1 ( Timestamp   := AxesGroup.State.SystemTime,
                            MessageType := MessageType.CMD,
                            Severity    := Severity.ERROR,
                            MessageCode := ErrorID,
                            MessageText := 'Invalid Parameter ParCmd.MoveTime = {1}',
                            Para1       := TIME_TO_STRING(ParCmd.MoveTime));
    RETURN;
  END_IF

  // Check ParCmd.BlendingMode valid ?
  IF (( ParCmd.OriMode <> OriMode.LINEAR_INTERPOLATED ) AND
      ( ParCmd.OriMode <> OriMode.JOINT_INTERPOLATED  ) AND
      ( ParCmd.OriMode <> OriMode.FIX                 ) AND
      ( ParCmd.OriMode <> OriMode.PATH                ))
  THEN
    // Parameter not valid
    CheckParameterValid := FALSE;
    // Set error
    ErrorID := RobotLibraryErrorIdEnum.ERR_INVALID_PAR_CMD;
    // Create log entry
    CreateLogMessagePara1 ( Timestamp   := AxesGroup.State.SystemTime,
                            MessageType := MessageType.CMD,
                            Severity    := Severity.ERROR,
                            MessageCode := ErrorID,
                            MessageText := 'Invalid Parameter ParCmd.OriMode = {1}',
                            Para1       := ORI_MODE_TO_STRING(ParCmd.OriMode));
    RETURN;
  END_IF

  // Check ParCmd.ConfigMode.Shoulder valid ?
  IF (( ParCmd.ConfigMode.Shoulder <> ArmConfigShoulder.USE_CONFIG ) AND
      ( ParCmd.ConfigMode.Shoulder <> ArmConfigShoulder.SAME       ) AND
      ( ParCmd.ConfigMode.Shoulder <> ArmConfigShoulder.FREE       ) AND
      ( ParCmd.ConfigMode.Shoulder <> ArmConfigShoulder.BACK       ) AND
      ( ParCmd.ConfigMode.Shoulder <> ArmConfigShoulder.FRONT      ))
  THEN
    // Parameter not valid
    CheckParameterValid := FALSE;
    // Set error
    ErrorID := RobotLibraryErrorIdEnum.ERR_INVALID_PAR_CMD;
    // Create log entry
    CreateLogMessagePara1 ( Timestamp   := AxesGroup.State.SystemTime,
                            MessageType := MessageType.CMD,
                            Severity    := Severity.ERROR,
                            MessageCode := ErrorID,
                            MessageText := 'Invalid Parameter ParCmd.ConfigMode.Shoulder = {1}',
                            Para1       :=  ARM_CONFIG_SHOULDER_TO_STRING(ParCmd.ConfigMode.Shoulder));
    RETURN;
  END_IF

  // Check ParCmd.ConfigMode.Elbow valid ?
  IF (( ParCmd.ConfigMode.Elbow <> ArmConfigElbow.USE_CONFIG ) AND
      ( ParCmd.ConfigMode.Elbow <> ArmConfigElbow.SAME       ) AND
      ( ParCmd.ConfigMode.Elbow <> ArmConfigElbow.FREE       ) AND
      ( ParCmd.ConfigMode.Elbow <> ArmConfigElbow.DOWN       ) AND
      ( ParCmd.ConfigMode.Elbow <> ArmConfigElbow.UP         ))
  THEN
    // Parameter not valid
    CheckParameterValid := FALSE;
    // Set error
    ErrorID := RobotLibraryErrorIdEnum.ERR_INVALID_PAR_CMD;
    // Create log entry
    CreateLogMessagePara1 ( Timestamp   := AxesGroup.State.SystemTime,
                            MessageType := MessageType.CMD,
                            Severity    := Severity.ERROR,
                            MessageCode := ErrorID,
                            MessageText := 'Invalid Parameter ParCmd.ConfigMode.Elbow = {1}',
                            Para1       :=  ARM_CONFIG_ELBOW_TO_STRING(ParCmd.ConfigMode.Elbow));
    RETURN;
  END_IF

  // Check ParCmd.ConfigMode.Wrist valid ?
  IF (( ParCmd.ConfigMode.Wrist <> ArmConfigWrist.USE_CONFIG ) AND
      ( ParCmd.ConfigMode.Wrist <> ArmConfigWrist.SAME       ) AND
      ( ParCmd.ConfigMode.Wrist <> ArmConfigWrist.FREE       ) AND
      ( ParCmd.ConfigMode.Wrist <> ArmConfigWrist.FLIP       ) AND
      ( ParCmd.ConfigMode.Wrist <> ArmConfigWrist.NON_FLIP   ))
  THEN
    // Parameter not valid
    CheckParameterValid := FALSE;
    // Set error
    ErrorID := RobotLibraryErrorIdEnum.ERR_INVALID_PAR_CMD;
    // Create log entry
    CreateLogMessagePara1 ( Timestamp   := AxesGroup.State.SystemTime,
                            MessageType := MessageType.CMD,
                            Severity    := Severity.ERROR,
                            MessageCode := ErrorID,
                            MessageText := 'Invalid Parameter ParCmd.ConfigMode.Wrist = {1}',
                            Para1       :=  ARM_CONFIG_WRIST_TO_STRING(ParCmd.ConfigMode.Wrist));
    RETURN;
  END_IF

  // Check ParCmd.TurnMode valid ?
  IF (( ParCmd.TurnMode <> TurnMode.USE_TURN_NUMBER ) AND
      ( ParCmd.TurnMode <> TurnMode.SAME            ) AND
      ( ParCmd.TurnMode <> TurnMode.FREE            ))
  THEN
    // Parameter not valid
    CheckParameterValid := FALSE;
    // Set error
    ErrorID := RobotLibraryErrorIdEnum.ERR_INVALID_PAR_CMD;
    // Create log entry
    CreateLogMessagePara1 ( Timestamp   := AxesGroup.State.SystemTime,
                            MessageType := MessageType.CMD,
                            Severity    := Severity.ERROR,
                            MessageCode := ErrorID,
                            MessageText := 'Invalid Parameter ParCmd.TurnMode = {1}',
                            Para1       :=  TURN_MODE_TO_STRING(ParCmd.TurnMode));
    RETURN;
  END_IF

  // Check ParCmd.Manipulation
  // -> no plausibility check for boolean

  FOR _idx := 0 TO 3
  DO
    // Check ParCmd.EmitterID valid ?
    IF  (( ParCmd.EmitterID[_idx] < -127 ) OR
         ( ParCmd.EmitterID[_idx] >  127 ))
    THEN
      // Parameter not valid
      CheckParameterValid := FALSE;
      // Set error
      ErrorID := RobotLibraryErrorIdEnum.ERR_INVALID_PAR_CMD;
      // Create log entry
      CreateLogMessagePara2 ( Timestamp   := AxesGroup.State.SystemTime,
                              MessageType := MessageType.CMD,
                              Severity    := Severity.ERROR,
                              MessageCode := ErrorID,
                              MessageText := 'Invalid Parameter ParCmd.EmitterID[{2}] = {1}',
                              Para1       := SINT_TO_STRING(ParCmd.EmitterID[_idx]),
                              Para2       := DINT_TO_STRING(_idx));
      EXIT;
      RETURN;
    END_IF
  END_FOR

END_METHOD

METHOD INTERNAL CreateCommandPayload : RobotLibraryCommandDataFB
VAR_IN_OUT
  /// Robot assignment of function
  AxesGroup : AxesGroup;
END_VAR
VAR
  /// internal index for loops
 _idx          : DINT;
  /// Parameter count
 _parameterCnt : DINT;
END_VAR
// Table 6-326: Sent CMD payload (PLC to RC) of "MoveCircularAbsolute"
// --------------------------
// Header
// --------------------------
// --------------------------
// Datablock
// --------------------------
// Byte 00 : UINT  - Type HB
// Byte 01 :       - Type LB
// Byte 02 : USINT - Reserve | ExecutionMode
// Byte 03 : USINT - ParSeq  | Priority
// --------------------------
// Datablock
// --------------------------
// Byte 04 : SINT       - EmitterID[0]
// Byte 05 : SINT       - EmitterID[1]
// Byte 06 : SINT       - EmitterID[2]
// Byte 07 : SINT       - EmitterID[3]
// Byte 08 : SINT       - ListenerID
// Byte 09 : BYTE       - Reserved
// Byte 10 : UINT       - VelocityRate HW HB
// Byte 11 :            - VelocityRate HW LB
// Byte 12 : UINT       - AccelerationRate HW HB
// Byte 13 :            - AccelerationRate HW LB
// Byte 14 : UINT       - DecelerationRate HW HB
// Byte 15 :            - DecelerationRate HW LB
// Byte 16 : UINT       - JerkRate HW HB
// Byte 17 :            - JerkRate HW LB
// Byte 18 : USINT      - ToolNo
// Byte 19 : USINT      - FrameNo
// Byte 20 : USINT      - BlendingMode
// Byte 21 : USINT      - OriMode
// Byte 22 : REAL       - BlendingParameter[0] HW HB
// Byte 23 :            - BlendingParameter[0] HW LB
// Byte 24 :            - BlendingParameter[0] LW HB
// Byte 25 :            - BlendingParameter[0] LW LB
// Byte 26 : REAL       - BlendingParameter[1] HW HB
// Byte 27 :            - BlendingParameter[1] HW LB
// Byte 28 :            - BlendingParameter[1] LW HB
// Byte 29 :            - BlendingParameter[1] LW LB
// Byte 30 : REAL       - AuxPoint.X HW HB
// Byte 31 :            - AuxPoint.X HW LB
// Byte 32 :            - AuxPoint.X LW HB
// Byte 33 :            - AuxPoint.X LW LB
// Byte 34 : REAL       - AuxPoint.Y HW HB
// Byte 35 :            - AuxPoint.Y HW LB
// Byte 36 :            - AuxPoint.Y LW HB
// Byte 37 :            - AuxPoint.Y LW LB
// Byte 38 : REAL       - AuxPoint.Z HW HB
// Byte 39 :            - AuxPoint.Z HW LB
// Byte 40 :            - AuxPoint.Z LW HB
// Byte 41 :            - AuxPoint.Z LW LB
// Byte 42 : REAL       - AuxPoint.RX HW HB
// Byte 43 :            - AuxPoint.RX HW LB
// Byte 44 :            - AuxPoint.RX LW HB
// Byte 45 :            - AuxPoint.RX LW LB
// Byte 46 : REAL       - AuxPoint.RY HW HB
// Byte 47 :            - AuxPoint.RY HW LB
// Byte 48 :            - AuxPoint.RY LW HB
// Byte 49 :            - AuxPoint.RY LW LB
// Byte 50 : REAL       - AuxPoint.RZ HW HB
// Byte 51 :            - AuxPoint.RZ HW LB
// Byte 52 :            - AuxPoint.RZ LW HB
// Byte 53 :            - AuxPoint.RZ LW LB
// Byte 54 : BYTE       - - - - - W E S
// Byte 55 : BYTE       - Reserved
// Byte 56 : BYTE       - AuxPoint.TurnNumber[0]
// Byte 57 : BYTE       - AuxPoint.TurnNumber[1]
// Byte 58 : BYTE       - AuxPoint.TurnNumber[2]
// Byte 59 : BYTE       - AuxPoint.TurnNumber[3]
// Byte 60 : REAL       - AuxPoint.E1 HW HB
// Byte 61 :            - AuxPoint.E1 HW LB
// Byte 62 :            - AuxPoint.E1 LW HB
// Byte 63 :            - AuxPoint.E1 LW LB
// Byte 64 : REAL       - EndPoint.X HW HB
// Byte 65 :            - EndPoint.X HW LB
// Byte 66 :            - EndPoint.X LW HB
// Byte 67 :            - EndPoint.X LW LB
// Byte 68 : REAL       - EndPoint.Y HW HB
// Byte 69 :            - EndPoint.Y HW LB
// Byte 70 :            - EndPoint.Y LW HB
// Byte 71 :            - EndPoint.Y LW LB
// Byte 72 : REAL       - EndPoint.Z HW HB
// Byte 73 :            - EndPoint.Z HW LB
// Byte 74 :            - EndPoint.Z LW HB
// Byte 75 :            - EndPoint.Z LW LB
// Byte 76 : REAL       - EndPoint.RX HW HB
// Byte 77 :            - EndPoint.RX HW LB
// Byte 78 :            - EndPoint.RX LW HB
// Byte 79 :            - EndPoint.RX LW LB
// Byte 80 : REAL       - EndPoint.RY HW HB
// Byte 81 :            - EndPoint.RY HW LB
// Byte 82 :            - EndPoint.RY LW HB
// Byte 83 :            - EndPoint.RY LW LB
// Byte 84 : REAL       - EndPoint.RZ HW HB
// Byte 85 :            - EndPoint.RZ HW LB
// Byte 86 :            - EndPoint.RZ LW HB
// Byte 87 :            - EndPoint.RZ LW LB
// Byte 88 : BYTE       - - - - - W E S
// Byte 89 : BYTE       - Reserved
// Byte 90 : BYTE       - EndPoint.TurnNumber[0]
// Byte 91 : BYTE       - EndPoint.TurnNumber[1]
// Byte 92 : BYTE       - EndPoint.TurnNumber[2]
// Byte 93 : BYTE       - EndPoint.TurnNumber[3]
// Byte 94 : REAL       - EndPoint.E1 HW HB
// Byte 95 :            - EndPoint.E1 HW LB
// Byte 96 :            - EndPoint.E1 LW HB
// Byte 97 :            - EndPoint.E1 LW LB
// Byte 98 : SINT       - CircMode
// Byte 99 : SINT       - CircPlane
// Byte 100: REAL       - Tolerance HW HB
// Byte 101:            - Tolerance HW LB
// Byte 102:            - Tolerance LW HB
// Byte 103:            - Tolerance LW LB
// Byte 104: REAL       - Angle HW HB
// Byte 105:            - Angle HW LB
// Byte 106:            - Angle LW HB
// Byte 107:            - Angle LW LB
// Byte 108: BOOL       - PathChoice
// Byte 109: BOOL       - Manipulation
// Byte 110: BYTE       - ConfigMode[0]
// Byte 111: BYTE       - ConfigMode[1]
// Byte 112: USINT      - TurnMode
// Byte 113: BYTE       - Reserved
// Byte 114: UINT       - Time HW HB
// Byte 115:            - Time HW LB
// Byte 116: REAL       - AuxPoint.E2 HW HB
// Byte 117:            - AuxPoint.E2 HW LB
// Byte 118:            - AuxPoint.E2 LW HB
// Byte 119:            - AuxPoint.E2 LW LB
// Byte 120: REAL       - AuxPoint.E3 HW HB
// Byte 121:            - AuxPoint.E3 HW LB
// Byte 122:            - AuxPoint.E3 LW HB
// Byte 123:            - AuxPoint.E3 LW LB
// Byte 124: REAL       - AuxPoint.E4 HW HB
// Byte 125:            - AuxPoint.E4 HW LB
// Byte 126:            - AuxPoint.E4 LW HB
// Byte 127:            - AuxPoint.E4 LW LB
// Byte 128: REAL       - AuxPoint.E5 HW HB
// Byte 129:            - AuxPoint.E5 HW LB
// Byte 130:            - AuxPoint.E5 LW HB
// Byte 131:            - AuxPoint.E5 LW LB
// Byte 132: REAL       - AuxPoint.E6 HW HB
// Byte 133:            - AuxPoint.E6 HW LB
// Byte 134:            - AuxPoint.E6 LW HB
// Byte 135:            - AuxPoint.E6 LW LB
// Byte 136: REAL       - EndPoint.E2 HW HB
// Byte 137:            - EndPoint.E2 HW LB
// Byte 138:            - EndPoint.E2 LW HB
// Byte 139:            - EndPoint.E2 LW LB
// Byte 140: REAL       - EndPoint.E3 HW HB
// Byte 141:            - EndPoint.E3 HW LB
// Byte 142:            - EndPoint.E3 LW HB
// Byte 143:            - EndPoint.E3 LW LB
// Byte 144: REAL       - EndPoint.E4 HW HB
// Byte 145:            - EndPoint.E4 HW LB
// Byte 146:            - EndPoint.E4 LW HB
// Byte 147:            - EndPoint.E4 LW LB
// Byte 148: REAL       - EndPoint.E5 HW HB
// Byte 149:            - EndPoint.E5 HW LB
// Byte 150:            - EndPoint.E5 LW HB
// Byte 151:            - EndPoint.E5 LW LB
// Byte 152: REAL       - EndPoint.E6 HW HB
// Byte 153:            - EndPoint.E6 HW LB
// Byte 154:            - EndPoint.E6 LW HB
// Byte 155:            - EndPoint.E6 LW LB

  // set command parameter
  _command.CmdTyp                    :=  CmdType.MoveCircularAbsolute;
  _command.ExecMode                  :=  ExecMode;
  _command.ParSeq                    := _command.ParSeq;
  _command.Priority                  :=  Priority;
  _command.EmitterID[0]              := _parCmd.EmitterID[0];
  _command.EmitterID[1]              := _parCmd.EmitterID[1];
  _command.EmitterID[2]              := _parCmd.EmitterID[2];
  _command.EmitterID[3]              := _parCmd.EmitterID[3];
  _command.ListenerID                := 0;
  _command.Reserve                   := 0;
  _command.VelocityRate              := REAL_TO_PERCENT_UINT(_parCmd.VelocityRate     , IsOptional := FALSE);
  _command.AccelerationRate          := REAL_TO_PERCENT_UINT(_parCmd.AccelerationRate , IsOptional := FALSE);
  _command.DecelerationRate          := REAL_TO_PERCENT_UINT(_parCmd.DecelerationRate , IsOptional := TRUE );
  _command.JerkRate                  := REAL_TO_PERCENT_UINT(_parCmd.JerkRate         , IsOptional := TRUE );
  _command.ToolNo                    := _parCmd.ToolNo;
  _command.FrameNo                   := _parCmd.FrameNo;
  _command.BlendingMode              := _parCmd.BlendingMode;
  _command.OriMode                   := _parCmd.OriMode;
  _command.BlendingParameter         := _parCmd.BlendingParameter;
  _command.AuxPoint                  := _parCmd.AuxPoint;
  _command.EndPoint                  := _parCmd.EndPoint;
  _command.CircMode                  := _parCmd.CircMode;
  _command.CircPlane                 := _parCmd.CircPlane;
  _command.Tolerance                 := _parCmd.Tolerance;
  _command.Angle                     := _parCmd.Angle;
  _command.PathChoice                := _parCmd.PathChoice.0;
  _command.Manipulation              := _parCmd.Manipulation;
  _command.ConfigMode                :=  ArmConfigParameterToBytes(_parCmd.ConfigMode);
  _command.TurnMode                  := _parCmd.TurnMode;
  _command.TurnMode                  := _parCmd.TurnMode;
  _command.MoveTime                  := TIME_TO_UINT(_parCmd.MoveTime);

  // copy command data to header
  _cmdHeader := _command;
  // call base implementation to copy header to payload buffer
  CreateCommandPayload := SUPER^.CreateCommandPayload(AxesGroup := AxesGroup);

  FOR _idx := 0 TO 3
  DO
    // Check parameter must be added ?
    IF ( CheckAddParameter(CreateCommandPayload.PayloadPtr))
    THEN
      // add command.EmitterID[x]
      CreateCommandPayload.AddSint(_command.EmitterID[_idx]);
      // inc parameter counter
     _parameterCnt := _parameterCnt + 1;
    END_IF
  END_FOR

  // Check parameter must be added ?
  IF ( CheckAddParameter(CreateCommandPayload.PayloadPtr))
  THEN
    // add command.ListenerID
    CreateCommandPayload.AddSint(_command.ListenerID);
    // inc parameter counter
   _parameterCnt := _parameterCnt + 1;
  END_IF

  // Check parameter must be added ?
  IF ( CheckAddParameter(CreateCommandPayload.PayloadPtr))
  THEN
    // add command.Reserve
    CreateCommandPayload.AddSint(_command.Reserve);
    // inc parameter counter
   _parameterCnt := _parameterCnt + 1;
  END_IF

  // Check parameter must be added ?
  IF ( CheckAddParameter(CreateCommandPayload.PayloadPtr))
  THEN
    // add command.VelocityRate
    CreateCommandPayload.AddUint(_command.VelocityRate);
    // inc parameter counter
   _parameterCnt := _parameterCnt + 1;
  END_IF

  // Check parameter must be added ?
  IF ( CheckAddParameter(CreateCommandPayload.PayloadPtr))
  THEN
    // add command.AccelerationRate
    CreateCommandPayload.AddUint(_command.AccelerationRate);
    // inc parameter counter
   _parameterCnt := _parameterCnt + 1;
  END_IF

  // Check parameter must be added ?
  IF ( CheckAddParameter(CreateCommandPayload.PayloadPtr))
  THEN
    // add command.DecelerationRate
    CreateCommandPayload.AddUint(_command.DecelerationRate);
    // inc parameter counter
   _parameterCnt := _parameterCnt + 1;
  END_IF

  // Check parameter must be added ?
  IF ( CheckAddParameter(CreateCommandPayload.PayloadPtr))
  THEN
    // add command.JerkRate
    CreateCommandPayload.AddUint(_command.JerkRate);
    // inc parameter counter
   _parameterCnt := _parameterCnt + 1;
  END_IF

  // Check parameter must be added ?
  IF ( CheckAddParameter(CreateCommandPayload.PayloadPtr))
  THEN
    // add command.ToolNo
    CreateCommandPayload.AddUsint(_command.ToolNo);
    // inc parameter counter
   _parameterCnt := _parameterCnt + 1;
  END_IF

  // Check parameter must be added ?
  IF ( CheckAddParameter(CreateCommandPayload.PayloadPtr))
  THEN
    // add command.mFrameNo
    CreateCommandPayload.AddUsint(_command.FrameNo);
    // inc parameter counter
   _parameterCnt := _parameterCnt + 1;
  END_IF

  // Check parameter must be added ?
  IF ( CheckAddParameter(CreateCommandPayload.PayloadPtr))
  THEN
    // add command.BlendingMode
    CreateCommandPayload.AddUsint(_command.BlendingMode);
    // inc parameter counter
   _parameterCnt := _parameterCnt + 1;
  END_IF

  // Check parameter must be added ?
  IF ( CheckAddParameter(CreateCommandPayload.PayloadPtr))
  THEN
    // add command.OriMode
    CreateCommandPayload.AddUsint(_command.OriMode);
    // inc parameter counter
   _parameterCnt := _parameterCnt + 1;
  END_IF

  // Check parameter must be added ?
  IF ( CheckAddParameter(CreateCommandPayload.PayloadPtr))
  THEN
    // add command.BlendingParameter[0]
    CreateCommandPayload.AddReal(_command.BlendingParameter[0]);
    // inc parameter counter
   _parameterCnt := _parameterCnt + 1;
  END_IF

  // Check parameter must be added ?
  IF ( CheckAddParameter(CreateCommandPayload.PayloadPtr))
  THEN
    // add command.BlendingParameter[1]
    CreateCommandPayload.AddReal(_command.BlendingParameter[1]);
    // inc parameter counter
   _parameterCnt := _parameterCnt + 1;
  END_IF

  // Check parameter must be added ?
  IF ( CheckAddParameter(CreateCommandPayload.PayloadPtr))
  THEN
    // add command.AuxPoint.X
    CreateCommandPayload.AddReal(_command.AuxPoint.X);
    // inc parameter counter
   _parameterCnt := _parameterCnt + 1;
  END_IF

  // Check parameter must be added ?
  IF ( CheckAddParameter(CreateCommandPayload.PayloadPtr))
  THEN
    // add command.AuxPoint.Y
    CreateCommandPayload.AddReal(_command.AuxPoint.Y);
    // inc parameter counter
   _parameterCnt := _parameterCnt + 1;
  END_IF

  // Check parameter must be added ?
  IF ( CheckAddParameter(CreateCommandPayload.PayloadPtr))
  THEN
    // add command.AuxPoint.Z
    CreateCommandPayload.AddReal(_command.AuxPoint.Z);
    // inc parameter counter
   _parameterCnt := _parameterCnt + 1;
  END_IF

  // Check parameter must be added ?
  IF ( CheckAddParameter(CreateCommandPayload.PayloadPtr))
  THEN
    // add command.AuxPoint.Rx
    CreateCommandPayload.AddReal(_command.AuxPoint.Rx);
    // inc parameter counter
   _parameterCnt := _parameterCnt + 1;
  END_IF

  // Check parameter must be added ?
  IF ( CheckAddParameter(CreateCommandPayload.PayloadPtr))
  THEN
    // add command.AuxPoint.Ry
    CreateCommandPayload.AddReal(_command.AuxPoint.Ry);
    // inc parameter counter
   _parameterCnt := _parameterCnt + 1;
  END_IF

  // Check parameter must be added ?
  IF ( CheckAddParameter(CreateCommandPayload.PayloadPtr))
  THEN
    // add command.AuxPoint.Rz
    CreateCommandPayload.AddReal(_command.AuxPoint.Rz);
    // inc parameter counter
   _parameterCnt := _parameterCnt + 1;
  END_IF

  // Check parameter must be added ?
  IF ( CheckAddParameter(CreateCommandPayload.PayloadPtr))
  THEN
    // add command.AuxPoint.Config
    CreateCommandPayload.AddArmConfig(_command.AuxPoint.Config);
    // inc parameter counter
   _parameterCnt := _parameterCnt + 1;
  END_IF

  // Check parameter must be added ?
  IF ( CheckAddParameter(CreateCommandPayload.PayloadPtr))
  THEN
    // add command.AuxPoint.TurnNumber
    CreateCommandPayload.AddTurnNumber(_command.AuxPoint.TurnNumber);
    // inc parameter counter
   _parameterCnt := _parameterCnt + 1;
  END_IF

  // Check parameter must be added ?
  IF ( CheckAddParameter(CreateCommandPayload.PayloadPtr))
  THEN
    // add command.AuxPoint.E1
    CreateCommandPayload.AddReal(_command.AuxPoint.E1);
    // inc parameter counter
   _parameterCnt := _parameterCnt + 1;
  END_IF

  // Check parameter must be added ?
  IF ( CheckAddParameter(CreateCommandPayload.PayloadPtr))
  THEN
    // add command.EndPoint.X
    CreateCommandPayload.AddReal(_command.EndPoint.X);
    // inc parameter counter
   _parameterCnt := _parameterCnt + 1;
  END_IF

  // Check parameter must be added ?
  IF ( CheckAddParameter(CreateCommandPayload.PayloadPtr))
  THEN
    // add command.EndPoint.Y
    CreateCommandPayload.AddReal(_command.EndPoint.y);
    // inc parameter counter
   _parameterCnt := _parameterCnt + 1;
  END_IF

  // Check parameter must be added ?
  IF ( CheckAddParameter(CreateCommandPayload.PayloadPtr))
  THEN
    // add command.EndPoint.Z
    CreateCommandPayload.AddReal(_command.EndPoint.Z);
    // inc parameter counter
   _parameterCnt := _parameterCnt + 1;
  END_IF

  // Check parameter must be added ?
  IF ( CheckAddParameter(CreateCommandPayload.PayloadPtr))
  THEN
    // add command.EndPoint.Rx
    CreateCommandPayload.AddReal(_command.EndPoint.Rx);
    // inc parameter counter
   _parameterCnt := _parameterCnt + 1;
  END_IF

  // Check parameter must be added ?
  IF ( CheckAddParameter(CreateCommandPayload.PayloadPtr))
  THEN
    // add command.EndPoint.Ry
    CreateCommandPayload.AddReal(_command.EndPoint.Ry);
    // inc parameter counter
   _parameterCnt := _parameterCnt + 1;
  END_IF

  // Check parameter must be added ?
  IF ( CheckAddParameter(CreateCommandPayload.PayloadPtr))
  THEN
    // add command.EndPoint.Rz
    CreateCommandPayload.AddReal(_command.EndPoint.Rz);
    // inc parameter counter
   _parameterCnt := _parameterCnt + 1;
  END_IF

  // Check parameter must be added ?
  IF ( CheckAddParameter(CreateCommandPayload.PayloadPtr))
  THEN
    // add command.EndPoint.Config
    CreateCommandPayload.AddArmConfig(_command.EndPoint.Config);
    // inc parameter counter
   _parameterCnt := _parameterCnt + 1;
  END_IF

  // Check parameter must be added ?
  IF ( CheckAddParameter(CreateCommandPayload.PayloadPtr))
  THEN
    // add command.EndPoint.TurnNumber
    CreateCommandPayload.AddTurnNumber(_command.EndPoint.TurnNumber);
    // inc parameter counter
   _parameterCnt := _parameterCnt + 1;
  END_IF

  // Check parameter must be added ?
  IF ( CheckAddParameter(CreateCommandPayload.PayloadPtr))
  THEN
    // add command.EndPoint.E1
    CreateCommandPayload.AddReal(_command.EndPoint.E1);
    // inc parameter counter
   _parameterCnt := _parameterCnt + 1;
  END_IF

  // Check parameter must be added ?
  IF ( CheckAddParameter(CreateCommandPayload.PayloadPtr))
  THEN
    // add command.CircMode
    CreateCommandPayload.AddSint(_command.CircMode);
    // inc parameter counter
   _parameterCnt := _parameterCnt + 1;
  END_IF

  // Check parameter must be added ?
  IF ( CheckAddParameter(CreateCommandPayload.PayloadPtr))
  THEN
    // add command.CircPlane
    CreateCommandPayload.AddSint(_command.CircPlane);
    // inc parameter counter
   _parameterCnt := _parameterCnt + 1;
  END_IF

  // Check parameter must be added ?
  IF ( CheckAddParameter(CreateCommandPayload.PayloadPtr))
  THEN
    // add command.Tolerance
    CreateCommandPayload.AddReal(_command.Tolerance);
    // inc parameter counter
   _parameterCnt := _parameterCnt + 1;
  END_IF

  // Check parameter must be added ?
  IF ( CheckAddParameter(CreateCommandPayload.PayloadPtr))
  THEN
    // add command.Angle
    CreateCommandPayload.AddReal(_command.Angle);
    // inc parameter counter
   _parameterCnt := _parameterCnt + 1;
  END_IF

  // Check parameter must be added ?
  IF ( CheckAddParameter(CreateCommandPayload.PayloadPtr))
  THEN
    // add command.PathChoice
    CreateCommandPayload.AddBool(_command.PathChoice);
    // inc parameter counter
   _parameterCnt := _parameterCnt + 1;
  END_IF

  // Check parameter must be added ?
  IF ( CheckAddParameter(CreateCommandPayload.PayloadPtr))
  THEN
    // add command.Manipulation
    CreateCommandPayload.AddBool(_command.Manipulation);
    // inc parameter counter
   _parameterCnt := _parameterCnt + 1;
  END_IF

  // Check parameter must be added ?
  IF ( CheckAddParameter(CreateCommandPayload.PayloadPtr))
  THEN
    // add command.Reserve2
    CreateCommandPayload.AddByte(_command.Reserve2);
    // inc parameter counter
   _parameterCnt := _parameterCnt + 1;
  END_IF

  // Check parameter must be added ?
  IF ( CheckAddParameter(CreateCommandPayload.PayloadPtr))
  THEN
    // add command.AuxPoint.E2
    CreateCommandPayload.AddReal(_command.AuxPoint.E2);
    // inc parameter counter
   _parameterCnt := _parameterCnt + 1;
  END_IF

  // Check parameter must be added ?
  IF ( CheckAddParameter(CreateCommandPayload.PayloadPtr))
  THEN
    // add command.AuxPoint.E3
    CreateCommandPayload.AddReal(_command.AuxPoint.E3);
    // inc parameter counter
   _parameterCnt := _parameterCnt + 1;
  END_IF

  // Check parameter must be added ?
  IF ( CheckAddParameter(CreateCommandPayload.PayloadPtr))
  THEN
    // add command.AuxPoint.E4
    CreateCommandPayload.AddReal(_command.AuxPoint.E4);
    // inc parameter counter
   _parameterCnt := _parameterCnt + 1;
  END_IF

  // Check parameter must be added ?
  IF ( CheckAddParameter(CreateCommandPayload.PayloadPtr))
  THEN
    // add command.AuxPoint.E5
    CreateCommandPayload.AddReal(_command.AuxPoint.E5);
    // inc parameter counter
   _parameterCnt := _parameterCnt + 1;
  END_IF

  // Check parameter must be added ?
  IF ( CheckAddParameter(CreateCommandPayload.PayloadPtr))
  THEN
    // add command.AuxPoint.E6
    CreateCommandPayload.AddReal(_command.AuxPoint.E6);
    // inc parameter counter
   _parameterCnt := _parameterCnt + 1;
  END_IF

  // Check parameter must be added ?
  IF ( CheckAddParameter(CreateCommandPayload.PayloadPtr))
  THEN
    // add command.EndPoint.E2
    CreateCommandPayload.AddReal(_command.EndPoint.E2);
    // inc parameter counter
   _parameterCnt := _parameterCnt + 1;
  END_IF

  // Check parameter must be added ?
  IF ( CheckAddParameter(CreateCommandPayload.PayloadPtr))
  THEN
    // add command.EndPoint.E3
    CreateCommandPayload.AddReal(_command.EndPoint.E3);
    // inc parameter counter
   _parameterCnt := _parameterCnt + 1;
  END_IF

  // Check parameter must be added ?
  IF ( CheckAddParameter(CreateCommandPayload.PayloadPtr))
  THEN
    // add command.EndPoint.E4
    CreateCommandPayload.AddReal(_command.EndPoint.E4);
    // inc parameter counter
   _parameterCnt := _parameterCnt + 1;
  END_IF

  // Check parameter must be added ?
  IF ( CheckAddParameter(CreateCommandPayload.PayloadPtr))
  THEN
    // add command.EndPoint.E5
    CreateCommandPayload.AddReal(_command.EndPoint.E5);
    // inc parameter counter
   _parameterCnt := _parameterCnt + 1;
  END_IF

  // Check parameter must be added ?
  IF ( CheckAddParameter(CreateCommandPayload.PayloadPtr))
  THEN
    // add command.EndPoint.E6
    CreateCommandPayload.AddReal(_command.EndPoint.E6);
    // inc parameter counter
   _parameterCnt := _parameterCnt + 1;
  END_IF

  // Create logging
  CreateCommandPayloadLog(AxesGroup := AxesGroup, ParameterCnt := _parameterCnt);

END_METHOD

METHOD INTERNAL CreateCommandPayloadLog
VAR_IN_OUT
  /// Robot assignment of function
  AxesGroup : AxesGroup;
END_VAR
VAR_INPUT
  /// Parameter count
  ParameterCnt : DINT;
END_VAR
VAR
  /// internal index for loops
 _idx : DINT;
END_VAR

  // Create log entry for Parameter start
  CreateLogMessagePara1 ( Timestamp   := AxesGroup.State.SystemTime,
                          MessageType := MessageType.CMD,
                          Severity    := Severity.DEBUG,
                          MessageCode := 0,
                          MessageText := 'Create command payload with the {1} parameter(s) :',
                          Para1       := DINT_TO_STRING(ParameterCnt));

  // Create log entry for EmitterID[x]
  FOR _idx := 0 TO 3
  DO
    // Return if no parameter is remaining...
    IF ( ParameterCnt = 0 ) THEN RETURN; END_IF
    // dec remaining parameter(s)
    ParameterCnt := ParameterCnt - 1;
    // Create log entry for Command.EmitterID
    CreateLogMessagePara2 ( Timestamp   := AxesGroup.State.SystemTime,
                            MessageType := MessageType.CMD,
                            Severity    := Severity.DEBUG,
                            MessageCode := 0,
                            MessageText := 'Command.EmitterID[{2}] = {1}',
                            Para1       :=  SINT_TO_STRING(_command.EmitterID[_idx]),
                            Para2       :=  DINT_TO_STRING(_idx));
  END_FOR

  // Return if no parameter is remaining...
  IF ( ParameterCnt = 0 ) THEN RETURN; END_IF
  // dec remaining parameter(s)
  ParameterCnt := ParameterCnt - 1;
  // Create log entry for ListenerID
  CreateLogMessagePara1 ( Timestamp   := AxesGroup.State.SystemTime,
                          MessageType := MessageType.CMD,
                          Severity    := Severity.DEBUG,
                          MessageCode := 0,
                          MessageText := 'Command.ListenerID = {1}',
                          Para1       :=  SINT_TO_STRING(_command.ListenerID));

  // Return if no parameter is remaining...
  IF ( ParameterCnt = 0 ) THEN RETURN; END_IF
  // dec remaining parameter(s)
  ParameterCnt := ParameterCnt - 1;
  // Create log entry for Reserve
  CreateLogMessagePara1 ( Timestamp   := AxesGroup.State.SystemTime,
                          MessageType := MessageType.CMD,
                          Severity    := Severity.DEBUG,
                          MessageCode := 0,
                          MessageText := 'Command.Reserve = {1}',
                          Para1       :=  SINT_TO_STRING(_command.Reserve));

  // Return if no parameter is remaining...
  IF ( ParameterCnt = 0 ) THEN RETURN; END_IF
  // dec remaining parameter(s)
  ParameterCnt := ParameterCnt - 1;
  // Create log entry for VelocityRate
  CreateLogMessagePara1 ( Timestamp   := AxesGroup.State.SystemTime,
                          MessageType := MessageType.CMD,
                          Severity    := Severity.DEBUG,
                          MessageCode := 0,
                          MessageText := 'Command.VelocityRate = {1}',
                          Para1       :=  UINT_TO_STRING(_command.VelocityRate));

  // Return if no parameter is remaining...
  IF ( ParameterCnt = 0 ) THEN RETURN; END_IF
  // dec remaining parameter(s)
  ParameterCnt := ParameterCnt - 1;
  // Create log entry for AccelerationRate
  CreateLogMessagePara1 ( Timestamp   := AxesGroup.State.SystemTime,
                          MessageType := MessageType.CMD,
                          Severity    := Severity.DEBUG,
                          MessageCode := 0,
                          MessageText := 'Command.AccelerationRate = {1}',
                          Para1       :=  UINT_TO_STRING(_command.AccelerationRate));

  // Return if no parameter is remaining...
  IF ( ParameterCnt = 0 ) THEN RETURN; END_IF
  // dec remaining parameter(s)
  ParameterCnt := ParameterCnt - 1;
  // Create log entry for DecelerationRate
  CreateLogMessagePara1 ( Timestamp   := AxesGroup.State.SystemTime,
                          MessageType := MessageType.CMD,
                          Severity    := Severity.DEBUG,
                          MessageCode := 0,
                          MessageText := 'Command.DecelerationRate = {1}',
                          Para1       :=  UINT_TO_STRING(_command.DecelerationRate));

  // Return if no parameter is remaining...
  IF ( ParameterCnt = 0 ) THEN RETURN; END_IF
  // dec remaining parameter(s)
  ParameterCnt := ParameterCnt - 1;
  // Create log entry for JerkRate
  CreateLogMessagePara1 ( Timestamp   := AxesGroup.State.SystemTime,
                          MessageType := MessageType.CMD,
                          Severity    := Severity.DEBUG,
                          MessageCode := 0,
                          MessageText := 'Command.JerkRate = {1}',
                          Para1       :=  UINT_TO_STRING(_command.JerkRate));

  // Return if no parameter is remaining...
  IF ( ParameterCnt = 0 ) THEN RETURN; END_IF
  // dec remaining parameter(s)
  ParameterCnt := ParameterCnt - 1;
  // Create log entry for ToolNo
  CreateLogMessagePara1 ( Timestamp   := AxesGroup.State.SystemTime,
                          MessageType := MessageType.CMD,
                          Severity    := Severity.DEBUG,
                          MessageCode := 0,
                          MessageText := 'Command.ToolNo = {1}',
                          Para1       :=  USINT_TO_STRING(_command.ToolNo));

  // Return if no parameter is remaining...
  IF ( ParameterCnt = 0 ) THEN RETURN; END_IF
  // dec remaining parameter(s)
  ParameterCnt := ParameterCnt - 1;
  // Create log entry for FrameNo
  CreateLogMessagePara1 ( Timestamp   := AxesGroup.State.SystemTime,
                          MessageType := MessageType.CMD,
                          Severity    := Severity.DEBUG,
                          MessageCode := 0,
                          MessageText := 'Command.FrameNo = {1}',
                          Para1       :=  USINT_TO_STRING(_command.FrameNo));

  // Return if no parameter is remaining...
  IF ( ParameterCnt = 0 ) THEN RETURN; END_IF
  // dec remaining parameter(s)
  ParameterCnt := ParameterCnt - 1;
  // Create log entry for BlendingMode
  CreateLogMessagePara1 ( Timestamp   := AxesGroup.State.SystemTime,
                          MessageType := MessageType.CMD,
                          Severity    := Severity.DEBUG,
                          MessageCode := 0,
                          MessageText := 'Command.BlendingMode = {1}',
                          Para1       :=  BLENDING_MODE_TO_STRING(_command.BlendingMode));

  // Return if no parameter is remaining...
  IF ( ParameterCnt = 0 ) THEN RETURN; END_IF
  // dec remaining parameter(s)
  ParameterCnt := ParameterCnt - 1;
  // Create log entry for OriMode
  CreateLogMessagePara1 ( Timestamp   := AxesGroup.State.SystemTime,
                          MessageType := MessageType.CMD,
                          Severity    := Severity.DEBUG,
                          MessageCode := 0,
                          MessageText := 'Command.OriMode = {1}',
                          Para1       :=  ORI_MODE_TO_STRING(_command.OriMode));

  // Return if no parameter is remaining...
  IF ( ParameterCnt = 0 ) THEN RETURN; END_IF
  // dec remaining parameter(s)
  ParameterCnt := ParameterCnt - 1;
  // Create log entry for BlendingParameter[0]
  CreateLogMessagePara1 ( Timestamp   := AxesGroup.State.SystemTime,
                          MessageType := MessageType.CMD,
                          Severity    := Severity.DEBUG,
                          MessageCode := 0,
                          MessageText := 'Command.BlendingParameter[0] = {1}',
                          Para1       :=  REAL_TO_STRING(_command.BlendingParameter[0]));

  // Return if no parameter is remaining...
  IF ( ParameterCnt = 0 ) THEN RETURN; END_IF
  // dec remaining parameter(s)
  ParameterCnt := ParameterCnt - 1;
  // Create log entry for BlendingParameter[1]
  CreateLogMessagePara1 ( Timestamp   := AxesGroup.State.SystemTime,
                          MessageType := MessageType.CMD,
                          Severity    := Severity.DEBUG,
                          MessageCode := 0,
                          MessageText := 'Command.BlendingParameter[1] = {1}',
                          Para1       :=  REAL_TO_STRING(_command.BlendingParameter[1]));

  // Return if no parameter is remaining...
  IF ( ParameterCnt = 0 ) THEN RETURN; END_IF
  // dec remaining parameter(s)
  ParameterCnt := ParameterCnt - 1;
  // Create log entry for AuxPoint.X
  CreateLogMessagePara1 ( Timestamp   := AxesGroup.State.SystemTime,
                          MessageType := MessageType.CMD,
                          Severity    := Severity.DEBUG,
                          MessageCode := 0,
                          MessageText := 'Command.AuxPoint.X = {1}',
                          Para1       :=  REAL_TO_STRING(_command.AuxPoint.X));

  // Return if no parameter is remaining...
  IF ( ParameterCnt = 0 ) THEN RETURN; END_IF
  // dec remaining parameter(s)
  ParameterCnt := ParameterCnt - 1;
  // Create log entry for AuxPoint.Y
  CreateLogMessagePara1 ( Timestamp   := AxesGroup.State.SystemTime,
                          MessageType := MessageType.CMD,
                          Severity    := Severity.DEBUG,
                          MessageCode := 0,
                          MessageText := 'Command.AuxPoint.Y = {1}',
                          Para1       :=  REAL_TO_STRING(_command.AuxPoint.Y));

  // Return if no parameter is remaining...
  IF ( ParameterCnt = 0 ) THEN RETURN; END_IF
  // dec remaining parameter(s)
  ParameterCnt := ParameterCnt - 1;
  // Create log entry for AuxPoint.Z
  CreateLogMessagePara1 ( Timestamp   := AxesGroup.State.SystemTime,
                          MessageType := MessageType.CMD,
                          Severity    := Severity.DEBUG,
                          MessageCode := 0,
                          MessageText := 'Command.AuxPoint.Z = {1}',
                          Para1       :=  REAL_TO_STRING(_command.AuxPoint.Z));

  // Return if no parameter is remaining...
  IF ( ParameterCnt = 0 ) THEN RETURN; END_IF
  // dec remaining parameter(s)
  ParameterCnt := ParameterCnt - 1;
  // Create log entry for AuxPoint.Rx
  CreateLogMessagePara1 ( Timestamp   := AxesGroup.State.SystemTime,
                          MessageType := MessageType.CMD,
                          Severity    := Severity.DEBUG,
                          MessageCode := 0,
                          MessageText := 'Command.AuxPoint.Rx = {1}',
                          Para1       :=  REAL_TO_STRING(_command.AuxPoint.Rx));

  // Return if no parameter is remaining...
  IF ( ParameterCnt = 0 ) THEN RETURN; END_IF
  // dec remaining parameter(s)
  ParameterCnt := ParameterCnt - 1;
  // Create log entry for AuxPoint.Ry
  CreateLogMessagePara1 ( Timestamp   := AxesGroup.State.SystemTime,
                          MessageType := MessageType.CMD,
                          Severity    := Severity.DEBUG,
                          MessageCode := 0,
                          MessageText := 'Command.AuxPoint.Ry = {1}',
                          Para1       :=  REAL_TO_STRING(_command.AuxPoint.Ry));

  // Return if no parameter is remaining...
  IF ( ParameterCnt = 0 ) THEN RETURN; END_IF
  // dec remaining parameter(s)
  ParameterCnt := ParameterCnt - 1;
  // Create log entry for AuxPoint.Rz
  CreateLogMessagePara1 ( Timestamp   := AxesGroup.State.SystemTime,
                          MessageType := MessageType.CMD,
                          Severity    := Severity.DEBUG,
                          MessageCode := 0,
                          MessageText := 'Command.AuxPoint.Rz = {1}',
                          Para1       :=  REAL_TO_STRING(_command.AuxPoint.Rz));

  // Return if no parameter is remaining...
  IF ( ParameterCnt = 0 ) THEN RETURN; END_IF
  // dec remaining parameter(s)
  ParameterCnt := ParameterCnt - 1;
  // Create log entry for AuxPoint.Config
  CreateLogMessagePara1 ( Timestamp   := AxesGroup.State.SystemTime,
                          MessageType := MessageType.CMD,
                          Severity    := Severity.DEBUG,
                          MessageCode := 0,
                          MessageText := 'Command.AuxPoint.Config = {1}',
                          Para1       :=  ARM_CONFIG_TO_STRING(_command.AuxPoint.Config));

  // Return if no parameter is remaining...
  IF ( ParameterCnt = 0 ) THEN RETURN; END_IF
  // dec remaining parameter(s)
  ParameterCnt := ParameterCnt - 1;
  // Create log entry for AuxPoint.Reserve
  CreateLogMessagePara1 ( Timestamp   := AxesGroup.State.SystemTime,
                          MessageType := MessageType.CMD,
                          Severity    := Severity.DEBUG,
                          MessageCode := 0,
                          MessageText := 'Command.AuxPoint.Config = {1}',
                          Para1       :=  SINT_TO_STRING(_command.Reserve));

  // Return if no parameter is remaining...
  IF ( ParameterCnt = 0 ) THEN RETURN; END_IF
  // dec remaining parameter(s)
  ParameterCnt := ParameterCnt - 1;
  // Create log entry for AuxPoint.TurnNumber[0]
  CreateLogMessagePara1 ( Timestamp   := AxesGroup.State.SystemTime,
                          MessageType := MessageType.CMD,
                          Severity    := Severity.DEBUG,
                          MessageCode := 0,
                          MessageText := 'Command.AuxPoint.TurnNumber[0] = {1}',
                          Para1       :=  BYTE_TO_STRING(CombineHalfSints(HalfSintHi := _command.AuxPoint.TurnNumber.J2Turns,
                                                                          HalfSintLo := _command.AuxPoint.TurnNumber.J1Turns)));

  // Return if no parameter is remaining...
  IF ( ParameterCnt = 0 ) THEN RETURN; END_IF
  // dec remaining parameter(s)
  ParameterCnt := ParameterCnt - 1;
  // Create log entry for AuxPoint.TurnNumber[1]
  CreateLogMessagePara1 ( Timestamp   := AxesGroup.State.SystemTime,
                          MessageType := MessageType.CMD,
                          Severity    := Severity.DEBUG,
                          MessageCode := 0,
                          MessageText := 'Command.AuxPoint.TurnNumber[1] = {1}',
                          Para1       :=  BYTE_TO_STRING(CombineHalfSints(HalfSintHi := _command.AuxPoint.TurnNumber.J4Turns,
                                                                          HalfSintLo := _command.AuxPoint.TurnNumber.J3Turns)));

  // Return if no parameter is remaining...
  IF ( ParameterCnt = 0 ) THEN RETURN; END_IF
  // dec remaining parameter(s)
  ParameterCnt := ParameterCnt - 1;
  // Create log entry for AuxPoint.TurnNumber[2]
  CreateLogMessagePara1 ( Timestamp   := AxesGroup.State.SystemTime,
                          MessageType := MessageType.CMD,
                          Severity    := Severity.DEBUG,
                          MessageCode := 0,
                          MessageText := 'Command.AuxPoint.TurnNumber[2] = {1}',
                          Para1       :=  BYTE_TO_STRING(CombineHalfSints(HalfSintHi := _command.AuxPoint.TurnNumber.J6Turns,
                                                                          HalfSintLo := _command.AuxPoint.TurnNumber.J5Turns)));

  // Return if no parameter is remaining...
  IF ( ParameterCnt = 0 ) THEN RETURN; END_IF
  // dec remaining parameter(s)
  ParameterCnt := ParameterCnt - 1;
  // Create log entry for AuxPoint.TurnNumber[3]
  CreateLogMessagePara1 ( Timestamp   := AxesGroup.State.SystemTime,
                          MessageType := MessageType.CMD,
                          Severity    := Severity.DEBUG,
                          MessageCode := 0,
                          MessageText := 'Command.AuxPoint.TurnNumber[3] = {1}',
                          Para1       :=  SINT_TO_STRING(_command.AuxPoint.TurnNumber.E1Turns));

  // Return if no parameter is remaining...
  IF ( ParameterCnt = 0 ) THEN RETURN; END_IF
  // dec remaining parameter(s)
  ParameterCnt := ParameterCnt - 1;
  // Create log entry for AuxPoint.E1
  CreateLogMessagePara1 ( Timestamp   := AxesGroup.State.SystemTime,
                          MessageType := MessageType.CMD,
                          Severity    := Severity.DEBUG,
                          MessageCode := 0,
                          MessageText := 'Command.AuxPoint.E1 = {1}',
                          Para1       :=  REAL_TO_STRING(_command.AuxPoint.E1));

  // Return if no parameter is remaining...
  IF ( ParameterCnt = 0 ) THEN RETURN; END_IF
  // dec remaining parameter(s)
  ParameterCnt := ParameterCnt - 1;
  // Create log entry for EndPoint.X
  CreateLogMessagePara1 ( Timestamp   := AxesGroup.State.SystemTime,
                          MessageType := MessageType.CMD,
                          Severity    := Severity.DEBUG,
                          MessageCode := 0,
                          MessageText := 'Command.EndPoint.X = {1}',
                          Para1       :=  REAL_TO_STRING(_command.EndPoint.X));

  // Return if no parameter is remaining...
  IF ( ParameterCnt = 0 ) THEN RETURN; END_IF
  // dec remaining parameter(s)
  ParameterCnt := ParameterCnt - 1;
  // Create log entry for EndPoint.Y
  CreateLogMessagePara1 ( Timestamp   := AxesGroup.State.SystemTime,
                          MessageType := MessageType.CMD,
                          Severity    := Severity.DEBUG,
                          MessageCode := 0,
                          MessageText := 'Command.EndPoint.Y = {1}',
                          Para1       :=  REAL_TO_STRING(_command.EndPoint.Y));

  // Return if no parameter is remaining...
  IF ( ParameterCnt = 0 ) THEN RETURN; END_IF
  // dec remaining parameter(s)
  ParameterCnt := ParameterCnt - 1;
  // Create log entry for EndPoint.Z
  CreateLogMessagePara1 ( Timestamp   := AxesGroup.State.SystemTime,
                          MessageType := MessageType.CMD,
                          Severity    := Severity.DEBUG,
                          MessageCode := 0,
                          MessageText := 'Command.EndPoint.Z = {1}',
                          Para1       :=  REAL_TO_STRING(_command.EndPoint.Z));

  // Return if no parameter is remaining...
  IF ( ParameterCnt = 0 ) THEN RETURN; END_IF
  // dec remaining parameter(s)
  ParameterCnt := ParameterCnt - 1;
  // Create log entry for EndPoint.Rx
  CreateLogMessagePara1 ( Timestamp   := AxesGroup.State.SystemTime,
                          MessageType := MessageType.CMD,
                          Severity    := Severity.DEBUG,
                          MessageCode := 0,
                          MessageText := 'Command.EndPoint.Rx = {1}',
                          Para1       :=  REAL_TO_STRING(_command.EndPoint.Rx));

  // Return if no parameter is remaining...
  IF ( ParameterCnt = 0 ) THEN RETURN; END_IF
  // dec remaining parameter(s)
  ParameterCnt := ParameterCnt - 1;
  // Create log entry for EndPoint.Ry
  CreateLogMessagePara1 ( Timestamp   := AxesGroup.State.SystemTime,
                          MessageType := MessageType.CMD,
                          Severity    := Severity.DEBUG,
                          MessageCode := 0,
                          MessageText := 'Command.EndPoint.Ry = {1}',
                          Para1       :=  REAL_TO_STRING(_command.EndPoint.Ry));

  // Return if no parameter is remaining...
  IF ( ParameterCnt = 0 ) THEN RETURN; END_IF
  // dec remaining parameter(s)
  ParameterCnt := ParameterCnt - 1;
  // Create log entry for EndPoint.Rz
  CreateLogMessagePara1 ( Timestamp   := AxesGroup.State.SystemTime,
                          MessageType := MessageType.CMD,
                          Severity    := Severity.DEBUG,
                          MessageCode := 0,
                          MessageText := 'Command.EndPoint.Rz = {1}',
                          Para1       :=  REAL_TO_STRING(_command.EndPoint.Rz));

  // Return if no parameter is remaining...
  IF ( ParameterCnt = 0 ) THEN RETURN; END_IF
  // dec remaining parameter(s)
  ParameterCnt := ParameterCnt - 1;
  // Create log entry for EndPoint.Config
  CreateLogMessagePara1 ( Timestamp   := AxesGroup.State.SystemTime,
                          MessageType := MessageType.CMD,
                          Severity    := Severity.DEBUG,
                          MessageCode := 0,
                          MessageText := 'Command.EndPoint.Config = {1}',
                          Para1       :=  ARM_CONFIG_TO_STRING(_command.EndPoint.Config));

  // Return if no parameter is remaining...
  IF ( ParameterCnt = 0 ) THEN RETURN; END_IF
  // dec remaining parameter(s)
  ParameterCnt := ParameterCnt - 1;
  // Create log entry for EndPoint.Reserve
  CreateLogMessagePara1 ( Timestamp   := AxesGroup.State.SystemTime,
                          MessageType := MessageType.CMD,
                          Severity    := Severity.DEBUG,
                          MessageCode := 0,
                          MessageText := 'Command.EndPoint.Config = {1}',
                          Para1       :=  SINT_TO_STRING(_command.Reserve));

  // Return if no parameter is remaining...
  IF ( ParameterCnt = 0 ) THEN RETURN; END_IF
  // dec remaining parameter(s)
  ParameterCnt := ParameterCnt - 1;
  // Create log entry for EndPoint.TurnNumber[0]
  CreateLogMessagePara1 ( Timestamp   := AxesGroup.State.SystemTime,
                          MessageType := MessageType.CMD,
                          Severity    := Severity.DEBUG,
                          MessageCode := 0,
                          MessageText := 'Command.EndPoint.TurnNumber[0] = {1}',
                          Para1       :=  BYTE_TO_STRING(CombineHalfSints(HalfSintHi := _command.EndPoint.TurnNumber.J2Turns,
                                                                          HalfSintLo := _command.EndPoint.TurnNumber.J1Turns)));

  // Return if no parameter is remaining...
  IF ( ParameterCnt = 0 ) THEN RETURN; END_IF
  // dec remaining parameter(s)
  ParameterCnt := ParameterCnt - 1;
  // Create log entry for EndPoint.TurnNumber[1]
  CreateLogMessagePara1 ( Timestamp   := AxesGroup.State.SystemTime,
                          MessageType := MessageType.CMD,
                          Severity    := Severity.DEBUG,
                          MessageCode := 0,
                          MessageText := 'Command.AuxPoint.EndPoint[1] = {1}',
                          Para1       :=  BYTE_TO_STRING(CombineHalfSints(HalfSintHi := _command.EndPoint.TurnNumber.J4Turns,
                                                                          HalfSintLo := _command.EndPoint.TurnNumber.J3Turns)));

  // Return if no parameter is remaining...
  IF ( ParameterCnt = 0 ) THEN RETURN; END_IF
  // dec remaining parameter(s)
  ParameterCnt := ParameterCnt - 1;
  // Create log entry for EndPoint.TurnNumber[2]
  CreateLogMessagePara1 ( Timestamp   := AxesGroup.State.SystemTime,
                          MessageType := MessageType.CMD,
                          Severity    := Severity.DEBUG,
                          MessageCode := 0,
                          MessageText := 'Command.EndPoint.TurnNumber[2] = {1}',
                          Para1       :=  BYTE_TO_STRING(CombineHalfSints(HalfSintHi := _command.EndPoint.TurnNumber.J6Turns,
                                                                          HalfSintLo := _command.EndPoint.TurnNumber.J5Turns)));

  // Return if no parameter is remaining...
  IF ( ParameterCnt = 0 ) THEN RETURN; END_IF
  // dec remaining parameter(s)
  ParameterCnt := ParameterCnt - 1;
  // Create log entry for EndPoint.TurnNumber[3]
  CreateLogMessagePara1 ( Timestamp   := AxesGroup.State.SystemTime,
                          MessageType := MessageType.CMD,
                          Severity    := Severity.DEBUG,
                          MessageCode := 0,
                          MessageText := 'Command.EndPoint.TurnNumber[3] = {1}',
                          Para1       :=  SINT_TO_STRING(_command.EndPoint.TurnNumber.E1Turns));

  // Return if no parameter is remaining...
  IF ( ParameterCnt = 0 ) THEN RETURN; END_IF
  // dec remaining parameter(s)
  ParameterCnt := ParameterCnt - 1;
  // Create log entry for EndPoint.E1
  CreateLogMessagePara1 ( Timestamp   := AxesGroup.State.SystemTime,
                          MessageType := MessageType.CMD,
                          Severity    := Severity.DEBUG,
                          MessageCode := 0,
                          MessageText := 'Command.EndPoint.E1 = {1}',
                          Para1       :=  REAL_TO_STRING(_command.EndPoint.E1));

  // Return if no parameter is remaining...
  IF ( ParameterCnt = 0 ) THEN RETURN; END_IF
  // dec remaining parameter(s)
  ParameterCnt := ParameterCnt - 1;
  // Create log entry for CircMode
  CreateLogMessagePara1 ( Timestamp   := AxesGroup.State.SystemTime,
                          MessageType := MessageType.CMD,
                          Severity    := Severity.DEBUG,
                          MessageCode := 0,
                          MessageText := 'Command.CircMode = {1}',
                          Para1       :=  CIRC_MODE_TO_STRING(_command.CircMode));
